LIN {X 0,Y 410.242,Z 474.921,A -85,B 0,C 180,E1 -10420.429,E2 -10420.429} C_VEL
LIN {X 0,Y 410.19,Z 477.706,A -85,B 0,C 180,E1 -10422.905,E2 -10422.905} C_VEL
LIN {X 0,Y 413.022,Z 490.224,A -85,B 0,C 180,E1 -10423.479,E2 -10423.479} C_VEL
LIN {X 0,Y 414.798,Z 499.639,A -85,B 0,C 180,E1 -10424.015,E2 -10424.015} C_VEL
LIN {X 0,Y 414.098,Z 513.044,A -85,B 0,C 180,E1 -10424.874,E2 -10424.874} C_VEL
LIN {X 0,Y 413.502,Z 524.652,A -85,B 0,C 180,E1 -10425.839,E2 -10425.839} C_VEL
LIN {X 0,Y 412.71,Z 536.519,A -85,B 0,C 180,E1 -10427.085,E2 -10427.085} C_VEL
LIN {X 0,Y 412.094,Z 545.096,A -85,B 0,C 180,E1 -10428.191,E2 -10428.191} C_VEL
LIN {X 0,Y 411.578,Z 553.045,A -85,B 0,C 180,E1 -10429.422,E2 -10429.422} C_VEL
LIN {X 0,Y 411.062,Z 560.821,A -85,B 0,C 180,E1 -10430.9,E2 -10430.9} C_VEL
LIN {X 0,Y 410.649,Z 568.02,A -85,B 0,C 180,E1 -10432.626,E2 -10432.626} C_VEL
LIN {X 0,Y 410.417,Z 572.805,A -85,B 0,C 180,E1 -10434.103,E2 -10434.103} C_VEL
LIN {X 0,Y 410.245,Z 576.463,A -85,B 0,C 180,E1 -10435.578,E2 -10435.578} C_VEL
LIN {X 0,Y 410.203,Z 579.083,A -85,B 0,C 180,E1 -10437.054,E2 -10437.054} C_VEL
LIN {X 0,Y 410.105,Z 580.298,A -85,B 0,C 180,E1 -10438.036,E2 -10438.036} C_VEL
LIN {X 0,Y 410.034,Z 581.469,A -85,B 0,C 180,E1 -10440,E2 -10440} C_VEL
LIN {X 0,Y 410.098,Z 581.463,A -85,B 0,C 180,E1 -10440.982,E2 -10440.982} C_VEL
LIN {X 0,Y 410.164,Z 581.016,A -85,B 0,C 180,E1 -10441.964,E2 -10441.964} C_VEL
LIN {X 0,Y 410.37,Z 578.907,A -85,B 0,C 180,E1 -10443.928,E2 -10443.928} C_VEL
LIN {X 0,Y 410.407,Z 576.222,A -85,B 0,C 180,E1 -10445.404,E2 -10445.404} C_VEL
LIN {X 0,Y 410.821,Z 571.701,A -85,B 0,C 180,E1 -10447.15,E2 -10447.15} C_VEL
LIN {X 0,Y 411.288,Z 565.724,A -85,B 0,C 180,E1 -10448.846,E2 -10448.846} C_VEL
LIN {X 0,Y 411.884,Z 559.118,A -85,B 0,C 180,E1 -10450.321,E2 -10450.321} C_VEL
LIN {X 0,Y 412.549,Z 550.966,A -85,B 0,C 180,E1 -10451.796,E2 -10451.796} C_VEL
LIN {X 0,Y 413.277,Z 542.616,A -85,B 0,C 180,E1 -10453.022,E2 -10453.022} C_VEL
LIN {X 0,Y 414.292,Z 531.763,A -85,B 0,C 180,E1 -10454.315,E2 -10454.315} C_VEL
LIN {X 0,Y 415.018,Z 521.116,A -85,B 0,C 180,E1 -10455.343,E2 -10455.343} C_VEL
LIN {X 0,Y 415.909,Z 508.281,A -85,B 0,C 180,E1 -10456.316,E2 -10456.316} C_VEL
LIN {X 0,Y 416.336,Z 500.964,A -85,B 0,C 180,E1 -10456.767,E2 -10456.767} C_VEL
LIN {X 0,Y 414.23,Z 492.241,A -85,B 0,C 180,E1 -10457.376,E2 -10457.376} C_VEL
LIN {X 0,Y 410.7,Z 481.456,A -85,B 0,C 180,E1 -10458.069,E2 -10458.069} C_VEL
LIN {X 0,Y 410.796,Z 479.163,A -85,B 0,C 180,E1 -10461.056,E2 -10461.056} C_VEL
LIN {X 0,Y 411.017,Z 476.941,A -85,B 0,C 180,E1 -10464.228,E2 -10464.228} C_VEL
LIN {X 0,Y 411.243,Z 474.906,A -85,B 0,C 180,E1 -10467.479,E2 -10467.479} C_VEL
LIN {X 0,Y 411.549,Z 473.168,A -85,B 0,C 180,E1 -10470.818,E2 -10470.818} C_VEL
LIN {X 0,Y 411.822,Z 472.142,A -85,B 0,C 180,E1 -10473.257,E2 -10473.257} C_VEL
LIN {X 0,Y 412.004,Z 471.503,A -85,B 0,C 180,E1 -10475.449,E2 -10475.449} C_VEL
LIN {X 0,Y 412.143,Z 471.083,A -85,B 0,C 180,E1 -10478.334,E2 -10478.334} C_VEL
LIN {X 0,Y 412.263,Z 471.372,A -85,B 0,C 180,E1 -10481.671,E2 -10481.671} C_VEL
LIN {X 0,Y 412.44,Z 472.28,A -85,B 0,C 180,E1 -10484.318,E2 -10484.318} C_VEL
LIN {X 0,Y 412.772,Z 473.906,A -85,B 0,C 180,E1 -10487.074,E2 -10487.074} C_VEL
LIN {X 0,Y 413.164,Z 476.415,A -85,B 0,C 180,E1 -10489.948,E2 -10489.948} C_VEL
LIN {X 0,Y 413.547,Z 479.076,A -85,B 0,C 180,E1 -10492.28,E2 -10492.28} C_VEL
LIN {X 0,Y 413.475,Z 482.47,A -85,B 0,C 180,E1 -10494.674,E2 -10494.674} C_VEL
LIN {X 0,Y 412.817,Z 487.359,A -85,B 0,C 180,E1 -10497.57,E2 -10497.57} C_VEL
LIN {X 0,Y 412.015,Z 493.889,A -85,B 0,C 180,E1 -10500.946,E2 -10500.946} C_VEL
LIN {X 0,Y 411.478,Z 500.74,A -85,B 0,C 180,E1 -10504.18,E2 -10504.18} C_VEL
LIN {X 0,Y 410.945,Z 509.273,A -85,B 0,C 180,E1 -10507.899,E2 -10507.899} C_VEL
LIN {X 0,Y 410.585,Z 516.838,A -85,B 0,C 180,E1 -10511.021,E2 -10511.021} C_VEL
LIN {X 0,Y 410.509,Z 518.931,A -85,B 0,C 180,E1 -10511.858,E2 -10511.858} C_VEL
LIN {X 0,Y 413.253,Z 533.559,A -85,B 0,C 180,E1 -10512.6,E2 -10512.6} C_VEL
LIN {X 0,Y 414.423,Z 546.638,A -85,B 0,C 180,E1 -10513.371,E2 -10513.371} C_VEL
LIN {X 0,Y 414.678,Z 554.233,A -85,B 0,C 180,E1 -10513.887,E2 -10513.887} C_VEL
LIN {X 0,Y 413.747,Z 566.78,A -85,B 0,C 180,E1 -10514.861,E2 -10514.861} C_VEL
LIN {X 0,Y 412.777,Z 578.942,A -85,B 0,C 180,E1 -10516.046,E2 -10516.046} C_VEL
LIN {X 0,Y 411.95,Z 588.41,A -85,B 0,C 180,E1 -10517.186,E2 -10517.186} C_VEL
LIN {X 0,Y 411.266,Z 598.435,A -85,B 0,C 180,E1 -10518.666,E2 -10518.666} C_VEL
LIN {X 0,Y 410.729,Z 606.584,A -85,B 0,C 180,E1 -10520.147,E2 -10520.147} C_VEL
LIN {X 0,Y 410.367,Z 613.151,A -85,B 0,C 180,E1 -10521.629,E2 -10521.629} C_VEL
LIN {X 0,Y 410.163,Z 618.42,A -85,B 0,C 180,E1 -10523.111,E2 -10523.111} C_VEL
LIN {X 0,Y 410.042,Z 622.525,A -85,B 0,C 180,E1 -10524.591,E2 -10524.591} C_VEL
LIN {X 0,Y 409.979,Z 625.565,A -85,B 0,C 180,E1 -10526.068,E2 -10526.068} C_VEL
LIN {X 0,Y 410.045,Z 627.027,A -85,B 0,C 180,E1 -10527.053,E2 -10527.053} C_VEL
LIN {X 0,Y 410.059,Z 628.075,A -85,B 0,C 180,E1 -10528.036,E2 -10528.036} C_VEL
LIN {X 0,Y 410.026,Z 628.699,A -85,B 0,C 180,E1 -10529.018,E2 -10529.018} C_VEL
LIN {X 0,Y 410.047,Z 628.867,A -85,B 0,C 180,E1 -10530,E2 -10530} C_VEL
LIN {X 0,Y 410.037,Z 628.623,A -85,B 0,C 180,E1 -10530.982,E2 -10530.982} C_VEL
LIN {X 0,Y 410.058,Z 627.976,A -85,B 0,C 180,E1 -10531.964,E2 -10531.964} C_VEL
LIN {X 0,Y 410.07,Z 626.896,A -85,B 0,C 180,E1 -10532.947,E2 -10532.947} C_VEL
LIN {X 0,Y 409.976,Z 625.339,A -85,B 0,C 180,E1 -10533.932,E2 -10533.932} C_VEL
LIN {X 0,Y 410.079,Z 622.192,A -85,B 0,C 180,E1 -10535.409,E2 -10535.409} C_VEL
LIN {X 0,Y 410.163,Z 617.933,A -85,B 0,C 180,E1 -10536.889,E2 -10536.889} C_VEL
LIN {X 0,Y 410.402,Z 611.438,A -85,B 0,C 180,E1 -10538.618,E2 -10538.618} C_VEL
LIN {X 0,Y 410.759,Z 604.31,A -85,B 0,C 180,E1 -10540.1,E2 -10540.1} C_VEL
LIN {X 0,Y 411.341,Z 595.431,A -85,B 0,C 180,E1 -10541.581,E2 -10541.581} C_VEL
LIN {X 0,Y 411.912,Z 586.362,A -85,B 0,C 180,E1 -10542.815,E2 -10542.815} C_VEL
LIN {X 0,Y 412.686,Z 575.411,A -85,B 0,C 180,E1 -10544.019,E2 -10544.019} C_VEL
LIN {X 0,Y 413.372,Z 563.98,A -85,B 0,C 180,E1 -10545.027,E2 -10545.027} C_VEL
LIN {X 0,Y 414.125,Z 551.921,A -85,B 0,C 180,E1 -10545.861,E2 -10545.861} C_VEL
LIN {X 0,Y 412.917,Z 539.848,A -85,B 0,C 180,E1 -10546.548,E2 -10546.548} C_VEL
LIN {X 0,Y 410.997,Z 525.799,A -85,B 0,C 180,E1 -10547.153,E2 -10547.153} C_VEL
LIN {X 0,Y 410.521,Z 522.375,A -85,B 0,C 180,E1 -10547.266,E2 -10547.266} C_VEL
LIN {X 0,Y 410.805,Z 514.358,A -85,B 0,C 180,E1 -10550.531,E2 -10550.531} C_VEL
LIN {X 0,Y 411.209,Z 506.721,A -85,B 0,C 180,E1 -10553.681,E2 -10553.681} C_VEL
LIN {X 0,Y 411.736,Z 499.086,A -85,B 0,C 180,E1 -10556.893,E2 -10556.893} C_VEL
LIN {X 0,Y 412.268,Z 491.444,A -85,B 0,C 180,E1 -10560.191,E2 -10560.191} C_VEL
LIN {X 0,Y 412.923,Z 483.99,A -85,B 0,C 180,E1 -10563.489,E2 -10563.489} C_VEL
LIN {X 0,Y 413.34,Z 478.666,A -85,B 0,C 180,E1 -10565.916,E2 -10565.916} C_VEL
LIN {X 0,Y 412.708,Z 473.491,A -85,B 0,C 180,E1 -10568.433,E2 -10568.433} C_VEL
LIN {X 0,Y 411.547,Z 466.979,A -85,B 0,C 180,E1 -10571.759,E2 -10571.759} C_VEL
LIN {X 0,Y 411.244,Z 465.261,A -85,B 0,C 180,E1 -10572.705,E2 -10572.705} C_VEL
LIN {X 0,Y 411.237,Z 465.262,A -85,B 0,C 180,E1 -10575.871,E2 -10575.871} C_VEL
LIN {X 0,Y 411.206,Z 465.265,A -85,B 0,C 180,E1 -10578.765,E2 -10578.765} C_VEL
LIN {X 0,Y 411.194,Z 465.264,A -85,B 0,C 180,E1 -10582.026,E2 -10582.026} C_VEL
LIN {X 0,Y 411.207,Z 465.262,A -85,B 0,C 180,E1 -10585.667,E2 -10585.667} C_VEL
LIN {X 0,Y 411.191,Z 465.265,A -85,B 0,C 180,E1 -10589.152,E2 -10589.152} C_VEL
LIN {X 0,Y 411.26,Z 465.258,A -85,B 0,C 180,E1 -10592.522,E2 -10592.522} C_VEL
LIN {X 0,Y 411.228,Z 465.258,A -85,B 0,C 180,E1 -10595.785,E2 -10595.785} C_VEL
LIN {X 0,Y 411.198,Z 465.266,A -85,B 0,C 180,E1 -10598.966,E2 -10598.966} C_VEL
LIN {X 0,Y 411.255,Z 465.257,A -85,B 0,C 180,E1 -10602.085,E2 -10602.085} C_VEL
LIN {X 0,Y 411.262,Z 465.257,A -85,B 0,C 180,E1 -10605.148,E2 -10605.148} C_VEL
LIN {X 0,Y 411.286,Z 465.254,A -85,B 0,C 180,E1 -10608.167,E2 -10608.167} C_VEL
LIN {X 0,Y 411.484,Z 465.23,A -85,B 0,C 180,E1 -10612.147,E2 -10612.147} C_VEL
LIN {X 0,Y 411.477,Z 465.231,A -85,B 0,C 180,E1 -10614.118,E2 -10614.118} C_VEL
LIN {X 0,Y 411.513,Z 465.225,A -85,B 0,C 180,E1 -10618.043,E2 -10618.043} C_VEL
LIN {X 0,Y 411.645,Z 465.21,A -85,B 0,C 180,E1 -10620,E2 -10620} C_VEL
LIN {X 0,Y 411.467,Z 465.231,A -85,B 0,C 180,E1 -10622.937,E2 -10622.937} C_VEL
LIN {X 0,Y 411.463,Z 465.232,A -85,B 0,C 180,E1 -10626.867,E2 -10626.867} C_VEL
LIN {X 0,Y 411.296,Z 465.252,A -85,B 0,C 180,E1 -10629.839,E2 -10629.839} C_VEL
LIN {X 0,Y 411.308,Z 465.25,A -85,B 0,C 180,E1 -10633.104,E2 -10633.104} C_VEL
LIN {X 0,Y 411.265,Z 465.257,A -85,B 0,C 180,E1 -10636.869,E2 -10636.869} C_VEL
LIN {X 0,Y 411.233,Z 465.261,A -85,B 0,C 180,E1 -10639.987,E2 -10639.987} C_VEL
LIN {X 0,Y 411.206,Z 465.263,A -85,B 0,C 180,E1 -10643.148,E2 -10643.148} C_VEL
LIN {X 0,Y 411.24,Z 465.262,A -85,B 0,C 180,E1 -10646.381,E2 -10646.381} C_VEL
LIN {X 0,Y 411.203,Z 465.264,A -85,B 0,C 180,E1 -10649.713,E2 -10649.713} C_VEL
LIN {X 0,Y 411.209,Z 465.26,A -85,B 0,C 180,E1 -10653.156,E2 -10653.156} C_VEL
LIN {X 0,Y 411.198,Z 465.266,A -85,B 0,C 180,E1 -10656.553,E2 -10656.553} C_VEL
LIN {X 0,Y 411.214,Z 465.262,A -85,B 0,C 180,E1 -10659.728,E2 -10659.728} C_VEL
LIN {X 0,Y 411.181,Z 465.266,A -85,B 0,C 180,E1 -10663.133,E2 -10663.133} C_VEL
LIN {X 0,Y 411.173,Z 465.268,A -85,B 0,C 180,E1 -10665.881,E2 -10665.881} C_VEL
LIN {X 0,Y 411.167,Z 465.268,A -85,B 0,C 180,E1 -10668.772,E2 -10668.772} C_VEL
LIN {X 0,Y 411.204,Z 465.265,A -85,B 0,C 180,E1 -10672.027,E2 -10672.027} C_VEL
LIN {X 0,Y 411.21,Z 465.262,A -85,B 0,C 180,E1 -10675.667,E2 -10675.667} C_VEL
LIN {X 0,Y 411.193,Z 465.264,A -85,B 0,C 180,E1 -10679.153,E2 -10679.153} C_VEL
LIN {X 0,Y 411.262,Z 465.256,A -85,B 0,C 180,E1 -10682.523,E2 -10682.523} C_VEL
LIN {X 0,Y 411.231,Z 465.262,A -85,B 0,C 180,E1 -10685.785,E2 -10685.785} C_VEL
LIN {X 0,Y 411.201,Z 465.262,A -85,B 0,C 180,E1 -10688.966,E2 -10688.966} C_VEL
LIN {X 0,Y 411.255,Z 465.259,A -85,B 0,C 180,E1 -10692.085,E2 -10692.085} C_VEL
LIN {X 0,Y 411.264,Z 465.255,A -85,B 0,C 180,E1 -10695.148,E2 -10695.148} C_VEL
LIN {X 0,Y 411.288,Z 465.255,A -85,B 0,C 180,E1 -10698.167,E2 -10698.167} C_VEL
LIN {X 0,Y 411.356,Z 465.244,A -85,B 0,C 180,E1 -10701.155,E2 -10701.155} C_VEL
LIN {X 0,Y 411.463,Z 465.234,A -85,B 0,C 180,E1 -10704.118,E2 -10704.118} C_VEL
LIN {X 0,Y 411.517,Z 465.226,A -85,B 0,C 180,E1 -10708.043,E2 -10708.043} C_VEL
LIN {X 0,Y 411.645,Z 465.211,A -85,B 0,C 180,E1 -10710,E2 -10710} C_VEL
LIN {X 0,Y 411.462,Z 465.23,A -85,B 0,C 180,E1 -10712.937,E2 -10712.937} C_VEL
LIN {X 0,Y 411.476,Z 465.231,A -85,B 0,C 180,E1 -10715.882,E2 -10715.882} C_VEL
LIN {X 0,Y 411.356,Z 465.243,A -85,B 0,C 180,E1 -10718.845,E2 -10718.845} C_VEL
LIN {X 0,Y 411.289,Z 465.254,A -85,B 0,C 180,E1 -10721.833,E2 -10721.833} C_VEL
LIN {X 0,Y 411.265,Z 465.254,A -85,B 0,C 180,E1 -10724.853,E2 -10724.853} C_VEL
LIN {X 0,Y 411.244,Z 465.257,A -85,B 0,C 180,E1 -10727.586,E2 -10727.586} C_VEL
LIN {X 0,Y 410.584,Z 465.343,A -85,B 0,C 180,E1 -10728.404,E2 -10728.404} C_VEL
LIN {X 0,Y 407.696,Z 465.704,A -85,B 0,C 180,E1 -10729.732,E2 -10729.732} C_VEL
LIN {X 0,Y 405.253,Z 466.005,A -85,B 0,C 180,E1 -10730.805,E2 -10730.805} C_VEL
LIN {X 0,Y 404.217,Z 466.135,A -85,B 0,C 180,E1 -10731.635,E2 -10731.635} C_VEL
LIN {X 0,Y 404.141,Z 466.14,A -85,B 0,C 180,E1 -10731.916,E2 -10731.916} C_VEL
LIN {X 0,Y 404.22,Z 466.134,A -85,B 0,C 180,E1 -10735.297,E2 -10735.297} C_VEL
LIN {X 0,Y 404.2,Z 466.139,A -85,B 0,C 180,E1 -10738,E2 -10738} C_VEL
LIN {X 0,Y 404.144,Z 466.145,A -85,B 0,C 180,E1 -10741.558,E2 -10741.558} C_VEL
LIN {X 0,Y 404.189,Z 466.137,A -85,B 0,C 180,E1 -10745.016,E2 -10745.016} C_VEL
LIN {X 0,Y 404.162,Z 466.139,A -85,B 0,C 180,E1 -10748.756,E2 -10748.756} C_VEL
LIN {X 0,Y 404.127,Z 466.146,A -85,B 0,C 180,E1 -10751.6,E2 -10751.6} C_VEL
LIN {X 0,Y 404.149,Z 466.14,A -85,B 0,C 180,E1 -10754.522,E2 -10754.522} C_VEL
LIN {X 0,Y 404.14,Z 466.145,A -85,B 0,C 180,E1 -10757.296,E2 -10757.296} C_VEL
LIN {X 0,Y 404.172,Z 466.142,A -85,B 0,C 180,E1 -10759.955,E2 -10759.955} C_VEL
LIN {X 0,Y 404.123,Z 466.145,A -85,B 0,C 180,E1 -10763.128,E2 -10763.128} C_VEL
LIN {X 0,Y 404.049,Z 466.154,A -85,B 0,C 180,E1 -10764.97,E2 -10764.97} C_VEL
LIN {X 0,Y 403.66,Z 466.204,A -85,B 0,C 180,E1 -10768.554,E2 -10768.554} C_VEL
LIN {X 0,Y 403.415,Z 466.238,A -85,B 0,C 180,E1 -10770.804,E2 -10770.804} C_VEL
LIN {X 0,Y 403.339,Z 468.056,A -85,B 0,C 180,E1 -10773.061,E2 -10773.061} C_VEL
LIN {X 0,Y 403.256,Z 470.252,A -85,B 0,C 180,E1 -10775.274,E2 -10775.274} C_VEL
LIN {X 0,Y 403.144,Z 473.565,A -85,B 0,C 180,E1 -10778.525,E2 -10778.525} C_VEL
LIN {X 0,Y 403.155,Z 475.779,A -85,B 0,C 180,E1 -10780.657,E2 -10780.657} C_VEL
LIN {X 0,Y 403.121,Z 477.917,A -85,B 0,C 180,E1 -10782.662,E2 -10782.662} C_VEL
LIN {X 0,Y 405.962,Z 490.643,A -85,B 0,C 180,E1 -10783.25,E2 -10783.25} C_VEL
LIN {X 0,Y 407.853,Z 500.898,A -85,B 0,C 180,E1 -10783.849,E2 -10783.849} C_VEL
LIN {X 0,Y 407.106,Z 514.287,A -85,B 0,C 180,E1 -10784.736,E2 -10784.736} C_VEL
LIN {X 0,Y 406.536,Z 525.173,A -85,B 0,C 180,E1 -10785.67,E2 -10785.67} C_VEL
LIN {X 0,Y 405.767,Z 536.345,A -85,B 0,C 180,E1 -10786.86,E2 -10786.86} C_VEL
LIN {X 0,Y 405.017,Z 546.743,A -85,B 0,C 180,E1 -10788.235,E2 -10788.235} C_VEL
LIN {X 0,Y 404.399,Z 555.835,A -85,B 0,C 180,E1 -10789.739,E2 -10789.739} C_VEL
LIN {X 0,Y 403.892,Z 563.194,A -85,B 0,C 180,E1 -10791.242,E2 -10791.242} C_VEL
LIN {X 0,Y 403.607,Z 568.167,A -85,B 0,C 180,E1 -10792.496,E2 -10792.496} C_VEL
LIN {X 0,Y 403.36,Z 573.012,A -85,B 0,C 180,E1 -10793.999,E2 -10793.999} C_VEL
LIN {X 0,Y 403.16,Z 576.726,A -85,B 0,C 180,E1 -10795.501,E2 -10795.501} C_VEL
LIN {X 0,Y 403.139,Z 579.398,A -85,B 0,C 180,E1 -10797.002,E2 -10797.002} C_VEL
LIN {X 0,Y 403.035,Z 580.663,A -85,B 0,C 180,E1 -10798.001,E2 -10798.001} C_VEL
LIN {X 0,Y 402.953,Z 581.89,A -85,B 0,C 180,E1 -10800,E2 -10800} C_VEL
LIN {X 0,Y 403.018,Z 581.912,A -85,B 0,C 180,E1 -10800.999,E2 -10800.999} C_VEL
LIN {X 0,Y 403.09,Z 581.508,A -85,B 0,C 180,E1 -10801.998,E2 -10801.998} C_VEL
LIN {X 0,Y 403.324,Z 579.443,A -85,B 0,C 180,E1 -10803.997,E2 -10803.997} C_VEL
LIN {X 0,Y 403.354,Z 576.8,A -85,B 0,C 180,E1 -10805.499,E2 -10805.499} C_VEL
LIN {X 0,Y 403.803,Z 572.489,A -85,B 0,C 180,E1 -10807.224,E2 -10807.224} C_VEL
LIN {X 0,Y 404.308,Z 566.458,A -85,B 0,C 180,E1 -10809,E2 -10809} C_VEL
LIN {X 0,Y 404.95,Z 559.945,A -85,B 0,C 180,E1 -10810.5,E2 -10810.5} C_VEL
LIN {X 0,Y 405.661,Z 551.887,A -85,B 0,C 180,E1 -10811.999,E2 -10811.999} C_VEL
LIN {X 0,Y 406.444,Z 543.623,A -85,B 0,C 180,E1 -10813.245,E2 -10813.245} C_VEL
LIN {X 0,Y 407.529,Z 532.805,A -85,B 0,C 180,E1 -10814.569,E2 -10814.569} C_VEL
LIN {X 0,Y 408.309,Z 522.565,A -85,B 0,C 180,E1 -10815.601,E2 -10815.601} C_VEL
LIN {X 0,Y 409.249,Z 510.108,A -85,B 0,C 180,E1 -10816.589,E2 -10816.589} C_VEL
LIN {X 0,Y 409.745,Z 502.76,A -85,B 0,C 180,E1 -10817.067,E2 -10817.067} C_VEL
LIN {X 0,Y 407.618,Z 493.899,A -85,B 0,C 180,E1 -10817.71,E2 -10817.71} C_VEL
LIN {X 0,Y 403.693,Z 482.076,A -85,B 0,C 180,E1 -10818.525,E2 -10818.525} C_VEL
LIN {X 0,Y 403.788,Z 479.932,A -85,B 0,C 180,E1 -10821.439,E2 -10821.439} C_VEL
LIN {X 0,Y 404.029,Z 477.77,A -85,B 0,C 180,E1 -10824.675,E2 -10824.675} C_VEL
LIN {X 0,Y 404.279,Z 475.811,A -85,B 0,C 180,E1 -10827.993,E2 -10827.993} C_VEL
LIN {X 0,Y 404.629,Z 474.173,A -85,B 0,C 180,E1 -10831.404,E2 -10831.404} C_VEL
LIN {X 0,Y 404.873,Z 473.332,A -85,B 0,C 180,E1 -10833.743,E2 -10833.743} C_VEL
LIN {X 0,Y 405.08,Z 472.757,A -85,B 0,C 180,E1 -10836.149,E2 -10836.149} C_VEL
LIN {X 0,Y 405.203,Z 472.55,A -85,B 0,C 180,E1 -10838.693,E2 -10838.693} C_VEL
LIN {X 0,Y 405.355,Z 472.927,A -85,B 0,C 180,E1 -10841.795,E2 -10841.795} C_VEL
LIN {X 0,Y 405.62,Z 474.313,A -85,B 0,C 180,E1 -10845.267,E2 -10845.267} C_VEL
LIN {X 0,Y 405.964,Z 476.262,A -85,B 0,C 180,E1 -10848.109,E2 -10848.109} C_VEL
LIN {X 0,Y 406.502,Z 479.632,A -85,B 0,C 180,E1 -10851.508,E2 -10851.508} C_VEL
LIN {X 0,Y 406.623,Z 481.2,A -85,B 0,C 180,E1 -10852.776,E2 -10852.776} C_VEL
LIN {X 0,Y 406.398,Z 484.692,A -85,B 0,C 180,E1 -10855.202,E2 -10855.202} C_VEL
LIN {X 0,Y 405.716,Z 489.579,A -85,B 0,C 180,E1 -10858.082,E2 -10858.082} C_VEL
LIN {X 0,Y 404.887,Z 496.099,A -85,B 0,C 180,E1 -10861.488,E2 -10861.488} C_VEL
LIN {X 0,Y 404.352,Z 502.758,A -85,B 0,C 180,E1 -10864.663,E2 -10864.663} C_VEL
LIN {X 0,Y 403.814,Z 511.578,A -85,B 0,C 180,E1 -10868.562,E2 -10868.562} C_VEL
LIN {X 0,Y 403.482,Z 518.346,A -85,B 0,C 180,E1 -10871.399,E2 -10871.399} C_VEL
LIN {X 0,Y 406.164,Z 531.761,A -85,B 0,C 180,E1 -10872.117,E2 -10872.117} C_VEL
LIN {X 0,Y 407.317,Z 542.322,A -85,B 0,C 180,E1 -10872.744,E2 -10872.744} C_VEL
LIN {X 0,Y 407.9,Z 554.877,A -85,B 0,C 180,E1 -10873.612,E2 -10873.612} C_VEL
LIN {X 0,Y 406.906,Z 567.099,A -85,B 0,C 180,E1 -10874.6,E2 -10874.6} C_VEL
LIN {X 0,Y 405.935,Z 578.273,A -85,B 0,C 180,E1 -10875.717,E2 -10875.717} C_VEL
LIN {X 0,Y 405.004,Z 588.378,A -85,B 0,C 180,E1 -10876.962,E2 -10876.962} C_VEL
LIN {X 0,Y 404.293,Z 598.314,A -85,B 0,C 180,E1 -10878.468,E2 -10878.468} C_VEL
LIN {X 0,Y 403.689,Z 606.372,A -85,B 0,C 180,E1 -10879.974,E2 -10879.974} C_VEL
LIN {X 0,Y 403.324,Z 612.89,A -85,B 0,C 180,E1 -10881.482,E2 -10881.482} C_VEL
LIN {X 0,Y 403.075,Z 618.117,A -85,B 0,C 180,E1 -10882.989,E2 -10882.989} C_VEL
LIN {X 0,Y 402.942,Z 622.187,A -85,B 0,C 180,E1 -10884.495,E2 -10884.495} C_VEL
LIN {X 0,Y 402.897,Z 625.201,A -85,B 0,C 180,E1 -10885.999,E2 -10885.999} C_VEL
LIN {X 0,Y 402.943,Z 626.649,A -85,B 0,C 180,E1 -10887.001,E2 -10887.001} C_VEL
LIN {X 0,Y 402.987,Z 627.685,A -85,B 0,C 180,E1 -10888.001,E2 -10888.001} C_VEL
LIN {X 0,Y 402.949,Z 628.281,A -85,B 0,C 180,E1 -10889.001,E2 -10889.001} C_VEL
LIN {X 0,Y 402.965,Z 628.432,A -85,B 0,C 180,E1 -10890,E2 -10890} C_VEL
LIN {X 0,Y 402.959,Z 628.174,A -85,B 0,C 180,E1 -10890.999,E2 -10890.999} C_VEL
LIN {X 0,Y 402.987,Z 627.511,A -85,B 0,C 180,E1 -10891.999,E2 -10891.999} C_VEL
LIN {X 0,Y 402.971,Z 626.39,A -85,B 0,C 180,E1 -10892.999,E2 -10892.999} C_VEL
LIN {X 0,Y 402.896,Z 624.815,A -85,B 0,C 180,E1 -10894.001,E2 -10894.001} C_VEL
LIN {X 0,Y 402.998,Z 621.622,A -85,B 0,C 180,E1 -10895.504,E2 -10895.504} C_VEL
LIN {X 0,Y 403.075,Z 617.312,A -85,B 0,C 180,E1 -10897.01,E2 -10897.01} C_VEL
LIN {X 0,Y 403.351,Z 610.761,A -85,B 0,C 180,E1 -10898.769,E2 -10898.769} C_VEL
LIN {X 0,Y 403.711,Z 603.543,A -85,B 0,C 180,E1 -10900.279,E2 -10900.279} C_VEL
LIN {X 0,Y 404.356,Z 594.597,A -85,B 0,C 180,E1 -10901.784,E2 -10901.784} C_VEL
LIN {X 0,Y 404.956,Z 585.444,A -85,B 0,C 180,E1 -10903.039,E2 -10903.039} C_VEL
LIN {X 0,Y 405.66,Z 575.352,A -85,B 0,C 180,E1 -10904.165,E2 -10904.165} C_VEL
LIN {X 0,Y 406.358,Z 564.32,A -85,B 0,C 180,E1 -10905.164,E2 -10905.164} C_VEL
LIN {X 0,Y 407.155,Z 552.212,A -85,B 0,C 180,E1 -10906.032,E2 -10906.032} C_VEL
LIN {X 0,Y 405.767,Z 538.968,A -85,B 0,C 180,E1 -10906.804,E2 -10906.804} C_VEL
LIN {X 0,Y 403.826,Z 525.012,A -85,B 0,C 180,E1 -10907.416,E2 -10907.416} C_VEL
LIN {X 0,Y 403.459,Z 522.002,A -85,B 0,C 180,E1 -10907.532,E2 -10907.532} C_VEL
LIN {X 0,Y 403.771,Z 513.899,A -85,B 0,C 180,E1 -10910.905,E2 -10910.905} C_VEL
LIN {X 0,Y 404.303,Z 505.031,A -85,B 0,C 180,E1 -10914.657,E2 -10914.657} C_VEL
LIN {X 0,Y 404.859,Z 497.426,A -85,B 0,C 180,E1 -10917.95,E2 -10917.95} C_VEL
LIN {X 0,Y 405.445,Z 489.784,A -85,B 0,C 180,E1 -10921.334,E2 -10921.334} C_VEL
LIN {X 0,Y 406.072,Z 483.349,A -85,B 0,C 180,E1 -10924.259,E2 -10924.259} C_VEL
LIN {X 0,Y 406.317,Z 479.589,A -85,B 0,C 180,E1 -10926.022,E2 -10926.022} C_VEL
LIN {X 0,Y 405.651,Z 474.386,A -85,B 0,C 180,E1 -10928.587,E2 -10928.587} C_VEL
LIN {X 0,Y 404.616,Z 468.458,A -85,B 0,C 180,E1 -10931.678,E2 -10931.678} C_VEL
LIN {X 0,Y 404.168,Z 466.142,A -85,B 0,C 180,E1 -10933.005,E2 -10933.005} C_VEL
LIN {X 0,Y 404.21,Z 466.137,A -85,B 0,C 180,E1 -10935.935,E2 -10935.935} C_VEL
LIN {X 0,Y 404.161,Z 466.142,A -85,B 0,C 180,E1 -10938.64,E2 -10938.64} C_VEL
LIN {X 0,Y 404.153,Z 466.14,A -85,B 0,C 180,E1 -10941.493,E2 -10941.493} C_VEL
LIN {X 0,Y 404.186,Z 466.14,A -85,B 0,C 180,E1 -10944.984,E2 -10944.984} C_VEL
LIN {X 0,Y 404.143,Z 466.146,A -85,B 0,C 180,E1 -10948.554,E2 -10948.554} C_VEL
LIN {X 0,Y 404.197,Z 466.136,A -85,B 0,C 180,E1 -10952,E2 -10952} C_VEL
LIN {X 0,Y 404.178,Z 466.137,A -85,B 0,C 180,E1 -10955.334,E2 -10955.334} C_VEL
LIN {X 0,Y 404.14,Z 466.145,A -85,B 0,C 180,E1 -10958.581,E2 -10958.581} C_VEL
LIN {X 0,Y 404.212,Z 466.133,A -85,B 0,C 180,E1 -10961.762,E2 -10961.762} C_VEL
LIN {X 0,Y 404.208,Z 466.136,A -85,B 0,C 180,E1 -10964.882,E2 -10964.882} C_VEL
LIN {X 0,Y 404.258,Z 466.129,A -85,B 0,C 180,E1 -10967.959,E2 -10967.959} C_VEL
LIN {X 0,Y 404.435,Z 466.108,A -85,B 0,C 180,E1 -10972.1,E2 -10972.1} C_VEL
LIN {X 0,Y 404.426,Z 466.109,A -85,B 0,C 180,E1 -10974.015,E2 -10974.015} C_VEL
LIN {X 0,Y 404.482,Z 466.1,A -85,B 0,C 180,E1 -10978.009,E2 -10978.009} C_VEL
LIN {X 0,Y 404.614,Z 466.085,A -85,B 0,C 180,E1 -10980,E2 -10980} C_VEL
LIN {X 0,Y 404.424,Z 466.108,A -85,B 0,C 180,E1 -10982.989,E2 -10982.989} C_VEL
LIN {X 0,Y 404.414,Z 466.11,A -85,B 0,C 180,E1 -10986.987,E2 -10986.987} C_VEL
LIN {X 0,Y 404.261,Z 466.129,A -85,B 0,C 180,E1 -10990.012,E2 -10990.012} C_VEL
LIN {X 0,Y 404.268,Z 466.126,A -85,B 0,C 180,E1 -10993.212,E2 -10993.212} C_VEL
LIN {X 0,Y 404.218,Z 466.133,A -85,B 0,C 180,E1 -10997.007,E2 -10997.007} C_VEL
LIN {X 0,Y 404.166,Z 466.143,A -85,B 0,C 180,E1 -11000.352,E2 -11000.352} C_VEL
LIN {X 0,Y 404.172,Z 466.139,A -85,B 0,C 180,E1 -11003.575,E2 -11003.575} C_VEL
LIN {X 0,Y 404.186,Z 466.137,A -85,B 0,C 180,E1 -11005.767,E2 -11005.767} C_VEL
LIN {X 0,Y 404.198,Z 466.138,A -85,B 0,C 180,E1 -11008,E2 -11008} C_VEL
LIN {X 0,Y 404.142,Z 466.142,A -85,B 0,C 180,E1 -11011.558,E2 -11011.558} C_VEL
LIN {X 0,Y 404.188,Z 466.137,A -85,B 0,C 180,E1 -11015.016,E2 -11015.016} C_VEL
LIN {X 0,Y 404.157,Z 466.142,A -85,B 0,C 180,E1 -11018.757,E2 -11018.757} C_VEL
LIN {X 0,Y 404.127,Z 466.144,A -85,B 0,C 180,E1 -11021.6,E2 -11021.6} C_VEL
LIN {X 0,Y 404.152,Z 466.144,A -85,B 0,C 180,E1 -11024.523,E2 -11024.523} C_VEL
LIN {X 0,Y 404.141,Z 466.141,A -85,B 0,C 180,E1 -11027.296,E2 -11027.296} C_VEL
LIN {X 0,Y 404.172,Z 466.142,A -85,B 0,C 180,E1 -11029.956,E2 -11029.956} C_VEL
LIN {X 0,Y 404.143,Z 466.142,A -85,B 0,C 180,E1 -11033.125,E2 -11033.125} C_VEL
LIN {X 0,Y 404.148,Z 466.145,A -85,B 0,C 180,E1 -11036.188,E2 -11036.188} C_VEL
LIN {X 0,Y 404.149,Z 466.143,A -85,B 0,C 180,E1 -11039.715,E2 -11039.715} C_VEL
LIN {X 0,Y 404.199,Z 466.134,A -85,B 0,C 180,E1 -11043.123,E2 -11043.123} C_VEL
LIN {X 0,Y 404.181,Z 466.138,A -85,B 0,C 180,E1 -11045.335,E2 -11045.335} C_VEL
LIN {X 0,Y 404.143,Z 466.143,A -85,B 0,C 180,E1 -11048.581,E2 -11048.581} C_VEL
LIN {X 0,Y 404.213,Z 466.136,A -85,B 0,C 180,E1 -11051.762,E2 -11051.762} C_VEL
LIN {X 0,Y 404.211,Z 466.133,A -85,B 0,C 180,E1 -11054.882,E2 -11054.882} C_VEL
LIN {X 0,Y 404.261,Z 466.132,A -85,B 0,C 180,E1 -11057.959,E2 -11057.959} C_VEL
LIN {X 0,Y 404.293,Z 466.123,A -85,B 0,C 180,E1 -11060.999,E2 -11060.999} C_VEL
LIN {X 0,Y 404.41,Z 466.113,A -85,B 0,C 180,E1 -11064.015,E2 -11064.015} C_VEL
LIN {X 0,Y 404.485,Z 466.102,A -85,B 0,C 180,E1 -11068.009,E2 -11068.009} C_VEL
LIN {X 0,Y 404.614,Z 466.087,A -85,B 0,C 180,E1 -11070,E2 -11070} C_VEL
LIN {X 0,Y 404.42,Z 466.107,A -85,B 0,C 180,E1 -11072.989,E2 -11072.989} C_VEL
LIN {X 0,Y 404.423,Z 466.11,A -85,B 0,C 180,E1 -11075.985,E2 -11075.985} C_VEL
LIN {X 0,Y 404.293,Z 466.122,A -85,B 0,C 180,E1 -11079.001,E2 -11079.001} C_VEL
LIN {X 0,Y 404.261,Z 466.13,A -85,B 0,C 180,E1 -11082.041,E2 -11082.041} C_VEL
LIN {X 0,Y 404.211,Z 466.133,A -85,B 0,C 180,E1 -11085.118,E2 -11085.118} C_VEL
LIN {X 0,Y 404.215,Z 466.135,A -85,B 0,C 180,E1 -11088.238,E2 -11088.238} C_VEL
LIN {X 0,Y 404.143,Z 466.143,A -85,B 0,C 180,E1 -11091.419,E2 -11091.419} C_VEL
LIN {X 0,Y 404.141,Z 466.14,A -85,B 0,C 180,E1 -11091.916,E2 -11091.916} C_VEL
LIN {X 0,Y 403.498,Z 466.222,A -85,B 0,C 180,E1 -11092.748,E2 -11092.748} C_VEL
LIN {X 0,Y 400.666,Z 466.579,A -85,B 0,C 180,E1 -11094.099,E2 -11094.099} C_VEL
LIN {X 0,Y 398.257,Z 466.882,A -85,B 0,C 180,E1 -11095.192,E2 -11095.192} C_VEL
LIN {X 0,Y 397.222,Z 467.008,A -85,B 0,C 180,E1 -11096.036,E2 -11096.036} C_VEL
LIN {X 0,Y 397.139,Z 467.017,A -85,B 0,C 180,E1 -11096.322,E2 -11096.322} C_VEL
LIN {X 0,Y 397.126,Z 467.016,A -85,B 0,C 180,E1 -11098.544,E2 -11098.544} C_VEL
LIN {X 0,Y 397.083,Z 467.024,A -85,B 0,C 180,E1 -11102.071,E2 -11102.071} C_VEL
LIN {X 0,Y 397.123,Z 467.018,A -85,B 0,C 180,E1 -11105.503,E2 -11105.503} C_VEL
LIN {X 0,Y 397.136,Z 467.014,A -85,B 0,C 180,E1 -11108.862,E2 -11108.862} C_VEL
LIN {X 0,Y 397.073,Z 467.024,A -85,B 0,C 180,E1 -11112.267,E2 -11112.267} C_VEL
LIN {X 0,Y 397.09,Z 467.02,A -85,B 0,C 180,E1 -11115.069,E2 -11115.069} C_VEL
LIN {X 0,Y 397.07,Z 467.026,A -85,B 0,C 180,E1 -11118.021,E2 -11118.021} C_VEL
LIN {X 0,Y 397.132,Z 467.016,A -85,B 0,C 180,E1 -11121.139,E2 -11121.139} C_VEL
LIN {X 0,Y 397.009,Z 467.031,A -85,B 0,C 180,E1 -11124.519,E2 -11124.519} C_VEL
LIN {X 0,Y 396.655,Z 467.079,A -85,B 0,C 180,E1 -11127.89,E2 -11127.89} C_VEL
LIN {X 0,Y 396.301,Z 467.127,A -85,B 0,C 180,E1 -11131.391,E2 -11131.391} C_VEL
LIN {X 0,Y 396.215,Z 470.434,A -85,B 0,C 180,E1 -11134.804,E2 -11134.804} C_VEL
LIN {X 0,Y 396.097,Z 473.785,A -85,B 0,C 180,E1 -11138.123,E2 -11138.123} C_VEL
LIN {X 0,Y 396.112,Z 476.028,A -85,B 0,C 180,E1 -11140.299,E2 -11140.299} C_VEL
LIN {X 0,Y 396.049,Z 478.389,A -85,B 0,C 180,E1 -11142.425,E2 -11142.425} C_VEL
LIN {X 0,Y 399.01,Z 491.767,A -85,B 0,C 180,E1 -11143.066,E2 -11143.066} C_VEL
LIN {X 0,Y 400.914,Z 501.376,A -85,B 0,C 180,E1 -11143.649,E2 -11143.649} C_VEL
LIN {X 0,Y 400.207,Z 513.572,A -85,B 0,C 180,E1 -11144.466,E2 -11144.466} C_VEL
LIN {X 0,Y 399.539,Z 525.667,A -85,B 0,C 180,E1 -11145.511,E2 -11145.511} C_VEL
LIN {X 0,Y 398.743,Z 537.091,A -85,B 0,C 180,E1 -11146.754,E2 -11146.754} C_VEL
LIN {X 0,Y 398.036,Z 546.584,A -85,B 0,C 180,E1 -11148.026,E2 -11148.026} C_VEL
LIN {X 0,Y 397.399,Z 555.777,A -85,B 0,C 180,E1 -11149.556,E2 -11149.556} C_VEL
LIN {X 0,Y 396.874,Z 563.226,A -85,B 0,C 180,E1 -11151.086,E2 -11151.086} C_VEL
LIN {X 0,Y 396.545,Z 568.276,A -85,B 0,C 180,E1 -11152.361,E2 -11152.361} C_VEL
LIN {X 0,Y 396.304,Z 573.194,A -85,B 0,C 180,E1 -11153.892,E2 -11153.892} C_VEL
LIN {X 0,Y 396.081,Z 576.976,A -85,B 0,C 180,E1 -11155.42,E2 -11155.42} C_VEL
LIN {X 0,Y 396.076,Z 579.709,A -85,B 0,C 180,E1 -11156.948,E2 -11156.948} C_VEL
LIN {X 0,Y 395.967,Z 581.018,A -85,B 0,C 180,E1 -11157.966,E2 -11157.966} C_VEL
LIN {X 0,Y 395.89,Z 581.867,A -85,B 0,C 180,E1 -11158.983,E2 -11158.983} C_VEL
LIN {X 0,Y 395.94,Z 582.36,A -85,B 0,C 180,E1 -11161.017,E2 -11161.017} C_VEL
LIN {X 0,Y 396.018,Z 581.999,A -85,B 0,C 180,E1 -11162.034,E2 -11162.034} C_VEL
LIN {X 0,Y 396.278,Z 579.992,A -85,B 0,C 180,E1 -11164.068,E2 -11164.068} C_VEL
LIN {X 0,Y 396.308,Z 577.416,A -85,B 0,C 180,E1 -11165.597,E2 -11165.597} C_VEL
LIN {X 0,Y 396.777,Z 573.346,A -85,B 0,C 180,E1 -11167.289,E2 -11167.289} C_VEL
LIN {X 0,Y 397.166,Z 569.069,A -85,B 0,C 180,E1 -11168.651,E2 -11168.651} C_VEL
LIN {X 0,Y 397.82,Z 563.088,A -85,B 0,C 180,E1 -11170.175,E2 -11170.175} C_VEL
LIN {X 0,Y 398.502,Z 555.662,A -85,B 0,C 180,E1 -11171.701,E2 -11171.701} C_VEL
LIN {X 0,Y 399.32,Z 546.472,A -85,B 0,C 180,E1 -11173.226,E2 -11173.226} C_VEL
LIN {X 0,Y 400.472,Z 537.193,A -85,B 0,C 180,E1 -11174.462,E2 -11174.462} C_VEL
LIN {X 0,Y 401.384,Z 526.537,A -85,B 0,C 180,E1 -11175.63,E2 -11175.63} C_VEL
LIN {X 0,Y 402.343,Z 515.244,A -85,B 0,C 180,E1 -11176.621,E2 -11176.621} C_VEL
LIN {X 0,Y 403.1,Z 504.828,A -85,B 0,C 180,E1 -11177.357,E2 -11177.357} C_VEL
LIN {X 0,Y 402.161,Z 499.439,A -85,B 0,C 180,E1 -11177.771,E2 -11177.771} C_VEL
LIN {X 0,Y 398.394,Z 487.612,A -85,B 0,C 180,E1 -11178.67,E2 -11178.67} C_VEL
LIN {X 0,Y 396.691,Z 482.723,A -85,B 0,C 180,E1 -11179.032,E2 -11179.032} C_VEL
LIN {X 0,Y 396.888,Z 479.988,A -85,B 0,C 180,E1 -11182.956,E2 -11182.956} C_VEL
LIN {X 0,Y 397.123,Z 477.984,A -85,B 0,C 180,E1 -11186.259,E2 -11186.259} C_VEL
LIN {X 0,Y 397.316,Z 476.765,A -85,B 0,C 180,E1 -11188.528,E2 -11188.528} C_VEL
LIN {X 0,Y 397.726,Z 475.257,A -85,B 0,C 180,E1 -11192.013,E2 -11192.013} C_VEL
LIN {X 0,Y 397.964,Z 474.523,A -85,B 0,C 180,E1 -11194.41,E2 -11194.41} C_VEL
LIN {X 0,Y 398.2,Z 474.045,A -85,B 0,C 180,E1 -11197.418,E2 -11197.418} C_VEL
LIN {X 0,Y 398.356,Z 474.237,A -85,B 0,C 180,E1 -11200.751,E2 -11200.751} C_VEL
LIN {X 0,Y 398.536,Z 475.103,A -85,B 0,C 180,E1 -11203.696,E2 -11203.696} C_VEL
LIN {X 0,Y 398.857,Z 476.677,A -85,B 0,C 180,E1 -11206.591,E2 -11206.591} C_VEL
LIN {X 0,Y 399.214,Z 478.906,A -85,B 0,C 180,E1 -11209.355,E2 -11209.355} C_VEL
LIN {X 0,Y 399.64,Z 482.082,A -85,B 0,C 180,E1 -11212.313,E2 -11212.313} C_VEL
LIN {X 0,Y 399.542,Z 485.052,A -85,B 0,C 180,E1 -11214.516,E2 -11214.516} C_VEL
LIN {X 0,Y 398.984,Z 488.835,A -85,B 0,C 180,E1 -11216.903,E2 -11216.903} C_VEL
LIN {X 0,Y 398.238,Z 494.068,A -85,B 0,C 180,E1 -11219.853,E2 -11219.853} C_VEL
LIN {X 0,Y 397.484,Z 501.834,A -85,B 0,C 180,E1 -11223.766,E2 -11223.766} C_VEL
LIN {X 0,Y 396.842,Z 510.183,A -85,B 0,C 180,E1 -11227.619,E2 -11227.619} C_VEL
LIN {X 0,Y 396.463,Z 517.85,A -85,B 0,C 180,E1 -11230.923,E2 -11230.923} C_VEL
LIN {X 0,Y 399.354,Z 531.827,A -85,B 0,C 180,E1 -11231.705,E2 -11231.705} C_VEL
LIN {X 0,Y 400.629,Z 542.882,A -85,B 0,C 180,E1 -11232.401,E2 -11232.401} C_VEL
LIN {X 0,Y 401.123,Z 555.575,A -85,B 0,C 180,E1 -11233.327,E2 -11233.327} C_VEL
LIN {X 0,Y 400.089,Z 567.527,A -85,B 0,C 180,E1 -11234.331,E2 -11234.331} C_VEL
LIN {X 0,Y 399.068,Z 578.469,A -85,B 0,C 180,E1 -11235.466,E2 -11235.466} C_VEL
LIN {X 0,Y 398.073,Z 588.419,A -85,B 0,C 180,E1 -11236.731,E2 -11236.731} C_VEL
LIN {X 0,Y 397.326,Z 598.249,A -85,B 0,C 180,E1 -11238.263,E2 -11238.263} C_VEL
LIN {X 0,Y 396.654,Z 606.198,A -85,B 0,C 180,E1 -11239.794,E2 -11239.794} C_VEL
LIN {X 0,Y 396.283,Z 612.659,A -85,B 0,C 180,E1 -11241.33,E2 -11241.33} C_VEL
LIN {X 0,Y 396.002,Z 617.837,A -85,B 0,C 180,E1 -11242.863,E2 -11242.863} C_VEL
LIN {X 0,Y 395.849,Z 621.869,A -85,B 0,C 180,E1 -11244.396,E2 -11244.396} C_VEL
LIN {X 0,Y 395.817,Z 624.847,A -85,B 0,C 180,E1 -11245.927,E2 -11245.927} C_VEL
LIN {X 0,Y 395.843,Z 626.278,A -85,B 0,C 180,E1 -11246.947,E2 -11246.947} C_VEL
LIN {X 0,Y 395.915,Z 627.3,A -85,B 0,C 180,E1 -11247.965,E2 -11247.965} C_VEL
LIN {X 0,Y 395.874,Z 627.859,A -85,B 0,C 180,E1 -11248.983,E2 -11248.983} C_VEL
LIN {X 0,Y 395.886,Z 627.992,A -85,B 0,C 180,E1 -11250,E2 -11250} C_VEL
LIN {X 0,Y 395.883,Z 627.716,A -85,B 0,C 180,E1 -11251.017,E2 -11251.017} C_VEL
LIN {X 0,Y 395.917,Z 627.03,A -85,B 0,C 180,E1 -11252.034,E2 -11252.034} C_VEL
LIN {X 0,Y 395.875,Z 625.869,A -85,B 0,C 180,E1 -11253.053,E2 -11253.053} C_VEL
LIN {X 0,Y 395.878,Z 623.325,A -85,B 0,C 180,E1 -11254.582,E2 -11254.582} C_VEL
LIN {X 0,Y 395.914,Z 619.362,A -85,B 0,C 180,E1 -11256.24,E2 -11256.24} C_VEL
LIN {X 0,Y 396.057,Z 614.957,A -85,B 0,C 180,E1 -11257.648,E2 -11257.648} C_VEL
LIN {X 0,Y 396.412,Z 607.786,A -85,B 0,C 180,E1 -11259.439,E2 -11259.439} C_VEL
LIN {X 0,Y 396.852,Z 599.962,A -85,B 0,C 180,E1 -11260.975,E2 -11260.975} C_VEL
LIN {X 0,Y 397.471,Z 592.001,A -85,B 0,C 180,E1 -11262.25,E2 -11262.25} C_VEL
LIN {X 0,Y 398.182,Z 581.602,A -85,B 0,C 180,E1 -11263.615,E2 -11263.615} C_VEL
LIN {X 0,Y 398.999,Z 570.348,A -85,B 0,C 180,E1 -11264.797,E2 -11264.797} C_VEL
LIN {X 0,Y 399.786,Z 558.158,A -85,B 0,C 180,E1 -11265.812,E2 -11265.812} C_VEL
LIN {X 0,Y 400.109,Z 551.72,A -85,B 0,C 180,E1 -11266.257,E2 -11266.257} C_VEL
LIN {X 0,Y 398.696,Z 539.049,A -85,B 0,C 180,E1 -11267.015,E2 -11267.015} C_VEL
LIN {X 0,Y 396.868,Z 525.276,A -85,B 0,C 180,E1 -11267.637,E2 -11267.637} C_VEL
LIN {X 0,Y 396.375,Z 521.702,A -85,B 0,C 180,E1 -11267.776,E2 -11267.776} C_VEL
LIN {X 0,Y 396.736,Z 513.445,A -85,B 0,C 180,E1 -11271.294,E2 -11271.294} C_VEL
LIN {X 0,Y 397.302,Z 504.597,A -85,B 0,C 180,E1 -11275.122,E2 -11275.122} C_VEL
LIN {X 0,Y 397.902,Z 496.997,A -85,B 0,C 180,E1 -11278.482,E2 -11278.482} C_VEL
LIN {X 0,Y 398.589,Z 488.859,A -85,B 0,C 180,E1 -11282.183,E2 -11282.183} C_VEL
LIN {X 0,Y 399.147,Z 483.024,A -85,B 0,C 180,E1 -11284.907,E2 -11284.907} C_VEL
LIN {X 0,Y 399.21,Z 479.166,A -85,B 0,C 180,E1 -11286.767,E2 -11286.767} C_VEL
LIN {X 0,Y 398.191,Z 472.881,A -85,B 0,C 180,E1 -11290.007,E2 -11290.007} C_VEL
LIN {X 0,Y 397.158,Z 467.015,A -85,B 0,C 180,E1 -11293.215,E2 -11293.215} C_VEL
LIN {X 0,Y 397.165,Z 467.015,A -85,B 0,C 180,E1 -11296.511,E2 -11296.511} C_VEL
LIN {X 0,Y 397.115,Z 467.017,A -85,B 0,C 180,E1 -11299.552,E2 -11299.552} C_VEL
LIN {X 0,Y 397.1,Z 467.021,A -85,B 0,C 180,E1 -11303.005,E2 -11303.005} C_VEL
LIN {X 0,Y 397.119,Z 467.019,A -85,B 0,C 180,E1 -11306.282,E2 -11306.282} C_VEL
LIN {X 0,Y 397.106,Z 467.02,A -85,B 0,C 180,E1 -11310.135,E2 -11310.135} C_VEL
LIN {X 0,Y 397.196,Z 467.01,A -85,B 0,C 180,E1 -11312.61,E2 -11312.61} C_VEL
LIN {X 0,Y 397.134,Z 467.014,A -85,B 0,C 180,E1 -11315.982,E2 -11315.982} C_VEL
LIN {X 0,Y 397.14,Z 467.014,A -85,B 0,C 180,E1 -11319.705,E2 -11319.705} C_VEL
LIN {X 0,Y 397.183,Z 467.011,A -85,B 0,C 180,E1 -11322.845,E2 -11322.845} C_VEL
LIN {X 0,Y 397.23,Z 467.006,A -85,B 0,C 180,E1 -11326.703,E2 -11326.703} C_VEL
LIN {X 0,Y 397.22,Z 467.003,A -85,B 0,C 180,E1 -11329.809,E2 -11329.809} C_VEL
LIN {X 0,Y 397.366,Z 466.989,A -85,B 0,C 180,E1 -11332.888,E2 -11332.888} C_VEL
LIN {X 0,Y 397.256,Z 467.002,A -85,B 0,C 180,E1 -11334.925,E2 -11334.925} C_VEL
LIN {X 0,Y 397.451,Z 466.976,A -85,B 0,C 180,E1 -11337.973,E2 -11337.973} C_VEL
LIN {X 0,Y 397.583,Z 466.961,A -85,B 0,C 180,E1 -11340,E2 -11340} C_VEL
LIN {X 0,Y 397.382,Z 466.985,A -85,B 0,C 180,E1 -11343.042,E2 -11343.042} C_VEL
LIN {X 0,Y 397.366,Z 466.987,A -85,B 0,C 180,E1 -11347.112,E2 -11347.112} C_VEL
LIN {X 0,Y 397.22,Z 467.006,A -85,B 0,C 180,E1 -11350.191,E2 -11350.191} C_VEL
LIN {X 0,Y 397.228,Z 467.003,A -85,B 0,C 180,E1 -11353.321,E2 -11353.321} C_VEL
LIN {X 0,Y 397.184,Z 467.009,A -85,B 0,C 180,E1 -11357.155,E2 -11357.155} C_VEL
LIN {X 0,Y 397.105,Z 467.021,A -85,B 0,C 180,E1 -11360.73,E2 -11360.73} C_VEL
LIN {X 0,Y 397.135,Z 467.017,A -85,B 0,C 180,E1 -11364.018,E2 -11364.018} C_VEL
LIN {X 0,Y 397.197,Z 467.007,A -85,B 0,C 180,E1 -11367.39,E2 -11367.39} C_VEL
LIN {X 0,Y 397.081,Z 467.023,A -85,B 0,C 180,E1 -11370.883,E2 -11370.883} C_VEL
LIN {X 0,Y 397.129,Z 467.018,A -85,B 0,C 180,E1 -11374.493,E2 -11374.493} C_VEL
LIN {X 0,Y 397.106,Z 467.021,A -85,B 0,C 180,E1 -11378.275,E2 -11378.275} C_VEL
LIN {X 0,Y 397.091,Z 467.02,A -85,B 0,C 180,E1 -11380.909,E2 -11380.909} C_VEL
LIN {X 0,Y 397.106,Z 467.02,A -85,B 0,C 180,E1 -11383.648,E2 -11383.648} C_VEL
LIN {X 0,Y 397.106,Z 467.021,A -85,B 0,C 180,E1 -11386.521,E2 -11386.521} C_VEL
LIN {X 0,Y 397.117,Z 467.02,A -85,B 0,C 180,E1 -11390.423,E2 -11390.423} C_VEL
LIN {X 0,Y 397.112,Z 467.022,A -85,B 0,C 180,E1 -11394.266,E2 -11394.266} C_VEL
LIN {X 0,Y 397.118,Z 467.018,A -85,B 0,C 180,E1 -11396.727,E2 -11396.727} C_VEL
LIN {X 0,Y 397.128,Z 467.02,A -85,B 0,C 180,E1 -11400.296,E2 -11400.296} C_VEL
LIN {X 0,Y 397.198,Z 467.008,A -85,B 0,C 180,E1 -11402.61,E2 -11402.61} C_VEL
LIN {X 0,Y 397.137,Z 467.017,A -85,B 0,C 180,E1 -11405.982,E2 -11405.982} C_VEL
LIN {X 0,Y 397.143,Z 467.015,A -85,B 0,C 180,E1 -11409.705,E2 -11409.705} C_VEL
LIN {X 0,Y 397.186,Z 467.009,A -85,B 0,C 180,E1 -11412.845,E2 -11412.845} C_VEL
LIN {X 0,Y 397.233,Z 467.002,A -85,B 0,C 180,E1 -11416.703,E2 -11416.703} C_VEL
LIN {X 0,Y 397.222,Z 467.007,A -85,B 0,C 180,E1 -11419.809,E2 -11419.809} C_VEL
LIN {X 0,Y 397.322,Z 466.991,A -85,B 0,C 180,E1 -11422.888,E2 -11422.888} C_VEL
LIN {X 0,Y 397.253,Z 466.999,A -85,B 0,C 180,E1 -11424.925,E2 -11424.925} C_VEL
LIN {X 0,Y 397.454,Z 466.978,A -85,B 0,C 180,E1 -11427.973,E2 -11427.973} C_VEL
LIN {X 0,Y 397.584,Z 466.963,A -85,B 0,C 180,E1 -11430,E2 -11430} C_VEL
LIN {X 0,Y 397.38,Z 466.984,A -85,B 0,C 180,E1 -11433.042,E2 -11433.042} C_VEL
LIN {X 0,Y 397.373,Z 466.989,A -85,B 0,C 180,E1 -11436.092,E2 -11436.092} C_VEL
LIN {X 0,Y 397.256,Z 466.999,A -85,B 0,C 180,E1 -11439.162,E2 -11439.162} C_VEL
LIN {X 0,Y 397.224,Z 467.007,A -85,B 0,C 180,E1 -11442.258,E2 -11442.258} C_VEL
LIN {X 0,Y 397.184,Z 467.009,A -85,B 0,C 180,E1 -11445.392,E2 -11445.392} C_VEL
LIN {X 0,Y 397.167,Z 467.012,A -85,B 0,C 180,E1 -11448.573,E2 -11448.573} C_VEL
LIN {X 0,Y 397.097,Z 467.022,A -85,B 0,C 180,E1 -11451.91,E2 -11451.91} C_VEL
LIN {X 0,Y 397.157,Z 467.015,A -85,B 0,C 180,E1 -11455.512,E2 -11455.512} C_VEL
LIN {X 0,Y 397.139,Z 467.017,A -85,B 0,C 180,E1 -11456.322,E2 -11456.322} C_VEL
LIN {X 0,Y 396.469,Z 467.1,A -85,B 0,C 180,E1 -11457.168,E2 -11457.168} C_VEL
LIN {X 0,Y 393.594,Z 467.456,A -85,B 0,C 180,E1 -11458.544,E2 -11458.544} C_VEL
LIN {X 0,Y 391.156,Z 467.762,A -85,B 0,C 180,E1 -11459.655,E2 -11459.655} C_VEL
LIN {X 0,Y 390.104,Z 467.89,A -85,B 0,C 180,E1 -11460.515,E2 -11460.515} C_VEL
LIN {X 0,Y 390.016,Z 467.9,A -85,B 0,C 180,E1 -11460.806,E2 -11460.806} C_VEL
LIN {X 0,Y 390.072,Z 467.898,A -85,B 0,C 180,E1 -11464.025,E2 -11464.025} C_VEL
LIN {X 0,Y 390.049,Z 467.9,A -85,B 0,C 180,E1 -11467.551,E2 -11467.551} C_VEL
LIN {X 0,Y 390.06,Z 467.896,A -85,B 0,C 180,E1 -11470.821,E2 -11470.821} C_VEL
LIN {X 0,Y 390.058,Z 467.9,A -85,B 0,C 180,E1 -11473.886,E2 -11473.886} C_VEL
LIN {X 0,Y 390.061,Z 467.896,A -85,B 0,C 180,E1 -11476.79,E2 -11476.79} C_VEL
LIN {X 0,Y 390.06,Z 467.899,A -85,B 0,C 180,E1 -11479.56,E2 -11479.56} C_VEL
LIN {X 0,Y 390.04,Z 467.898,A -85,B 0,C 180,E1 -11482.45,E2 -11482.45} C_VEL
LIN {X 0,Y 389.929,Z 467.912,A -85,B 0,C 180,E1 -11484.776,E2 -11484.776} C_VEL
LIN {X 0,Y 389.556,Z 467.96,A -85,B 0,C 180,E1 -11488.453,E2 -11488.453} C_VEL
LIN {X 0,Y 389.307,Z 467.994,A -85,B 0,C 180,E1 -11490.829,E2 -11490.829} C_VEL
LIN {X 0,Y 389.215,Z 468.579,A -85,B 0,C 180,E1 -11492.226,E2 -11492.226} C_VEL
LIN {X 0,Y 389.074,Z 471.747,A -85,B 0,C 180,E1 -11495.451,E2 -11495.451} C_VEL
LIN {X 0,Y 389.007,Z 475.137,A -85,B 0,C 180,E1 -11498.818,E2 -11498.818} C_VEL
LIN {X 0,Y 388.952,Z 478.569,A -85,B 0,C 180,E1 -11502.144,E2 -11502.144} C_VEL
LIN {X 0,Y 392.368,Z 494.104,A -85,B 0,C 180,E1 -11502.948,E2 -11502.948} C_VEL
LIN {X 0,Y 393.942,Z 502.475,A -85,B 0,C 180,E1 -11503.481,E2 -11503.481} C_VEL
LIN {X 0,Y 393.251,Z 514.547,A -85,B 0,C 180,E1 -11504.317,E2 -11504.317} C_VEL
LIN {X 0,Y 392.562,Z 526.198,A -85,B 0,C 180,E1 -11505.35,E2 -11505.35} C_VEL
LIN {X 0,Y 391.73,Z 537.837,A -85,B 0,C 180,E1 -11506.644,E2 -11506.644} C_VEL
LIN {X 0,Y 391.045,Z 546.392,A -85,B 0,C 180,E1 -11507.809,E2 -11507.809} C_VEL
LIN {X 0,Y 390.376,Z 555.72,A -85,B 0,C 180,E1 -11509.366,E2 -11509.366} C_VEL
LIN {X 0,Y 389.834,Z 563.257,A -85,B 0,C 180,E1 -11510.924,E2 -11510.924} C_VEL
LIN {X 0,Y 389.488,Z 568.386,A -85,B 0,C 180,E1 -11512.222,E2 -11512.222} C_VEL
LIN {X 0,Y 389.249,Z 573.377,A -85,B 0,C 180,E1 -11513.781,E2 -11513.781} C_VEL
LIN {X 0,Y 389.008,Z 577.226,A -85,B 0,C 180,E1 -11515.337,E2 -11515.337} C_VEL
LIN {X 0,Y 388.995,Z 580.02,A -85,B 0,C 180,E1 -11516.893,E2 -11516.893} C_VEL
LIN {X 0,Y 388.901,Z 581.359,A -85,B 0,C 180,E1 -11517.929,E2 -11517.929} C_VEL
LIN {X 0,Y 388.817,Z 582.26,A -85,B 0,C 180,E1 -11518.964,E2 -11518.964} C_VEL
LIN {X 0,Y 388.865,Z 582.813,A -85,B 0,C 180,E1 -11521.035,E2 -11521.035} C_VEL
LIN {X 0,Y 388.95,Z 582.499,A -85,B 0,C 180,E1 -11522.071,E2 -11522.071} C_VEL
LIN {X 0,Y 389.06,Z 581.74,A -85,B 0,C 180,E1 -11523.106,E2 -11523.106} C_VEL
LIN {X 0,Y 389.233,Z 580.566,A -85,B 0,C 180,E1 -11524.142,E2 -11524.142} C_VEL
LIN {X 0,Y 389.265,Z 578.047,A -85,B 0,C 180,E1 -11525.699,E2 -11525.699} C_VEL
LIN {X 0,Y 389.76,Z 574.17,A -85,B 0,C 180,E1 -11527.368,E2 -11527.368} C_VEL
LIN {X 0,Y 390.194,Z 569.816,A -85,B 0,C 180,E1 -11528.806,E2 -11528.806} C_VEL
LIN {X 0,Y 390.889,Z 563.945,A -85,B 0,C 180,E1 -11530.358,E2 -11530.358} C_VEL
LIN {X 0,Y 391.624,Z 556.676,A -85,B 0,C 180,E1 -11531.91,E2 -11531.91} C_VEL
LIN {X 0,Y 392.5,Z 547.6,A -85,B 0,C 180,E1 -11533.46,E2 -11533.46} C_VEL
LIN {X 0,Y 393.701,Z 538.377,A -85,B 0,C 180,E1 -11534.724,E2 -11534.724} C_VEL
LIN {X 0,Y 394.751,Z 527.388,A -85,B 0,C 180,E1 -11535.971,E2 -11535.971} C_VEL
LIN {X 0,Y 395.842,Z 515.603,A -85,B 0,C 180,E1 -11537.035,E2 -11537.035} C_VEL
LIN {X 0,Y 396.564,Z 505.609,A -85,B 0,C 180,E1 -11537.764,E2 -11537.764} C_VEL
LIN {X 0,Y 394.524,Z 497.233,A -85,B 0,C 180,E1 -11538.451,E2 -11538.451} C_VEL
LIN {X 0,Y 390.745,Z 486.365,A -85,B 0,C 180,E1 -11539.321,E2 -11539.321} C_VEL
LIN {X 0,Y 389.72,Z 483.389,A -85,B 0,C 180,E1 -11539.557,E2 -11539.557} C_VEL
LIN {X 0,Y 389.899,Z 480.866,A -85,B 0,C 180,E1 -11543.363,E2 -11543.363} C_VEL
LIN {X 0,Y 390.162,Z 478.9,A -85,B 0,C 180,E1 -11546.765,E2 -11546.765} C_VEL
LIN {X 0,Y 390.384,Z 477.752,A -85,B 0,C 180,E1 -11549.083,E2 -11549.083} C_VEL
LIN {X 0,Y 390.805,Z 476.394,A -85,B 0,C 180,E1 -11552.65,E2 -11552.65} C_VEL
LIN {X 0,Y 391.058,Z 475.774,A -85,B 0,C 180,E1 -11555.106,E2 -11555.106} C_VEL
LIN {X 0,Y 391.287,Z 475.485,A -85,B 0,C 180,E1 -11557.786,E2 -11557.786} C_VEL
LIN {X 0,Y 391.421,Z 475.813,A -85,B 0,C 180,E1 -11561.052,E2 -11561.052} C_VEL
LIN {X 0,Y 391.682,Z 476.982,A -85,B 0,C 180,E1 -11564.41,E2 -11564.41} C_VEL
LIN {X 0,Y 392.015,Z 478.75,A -85,B 0,C 180,E1 -11567.311,E2 -11567.311} C_VEL
LIN {X 0,Y 392.407,Z 481.41,A -85,B 0,C 180,E1 -11570.366,E2 -11570.366} C_VEL
LIN {X 0,Y 392.699,Z 483.805,A -85,B 0,C 180,E1 -11572.52,E2 -11572.52} C_VEL
LIN {X 0,Y 392.457,Z 487.241,A -85,B 0,C 180,E1 -11575.037,E2 -11575.037} C_VEL
LIN {X 0,Y 391.706,Z 492.077,A -85,B 0,C 180,E1 -11578.042,E2 -11578.042} C_VEL
LIN {X 0,Y 390.972,Z 497.333,A -85,B 0,C 180,E1 -11580.965,E2 -11580.965} C_VEL
LIN {X 0,Y 390.324,Z 504.131,A -85,B 0,C 180,E1 -11584.397,E2 -11584.397} C_VEL
LIN {X 0,Y 389.702,Z 512.504,A -85,B 0,C 180,E1 -11588.302,E2 -11588.302} C_VEL
LIN {X 0,Y 389.446,Z 517.406,A -85,B 0,C 180,E1 -11590.394,E2 -11590.394} C_VEL
LIN {X 0,Y 392.384,Z 530.708,A -85,B 0,C 180,E1 -11591.192,E2 -11591.192} C_VEL
LIN {X 0,Y 393.928,Z 542.735,A -85,B 0,C 180,E1 -11591.989,E2 -11591.989} C_VEL
LIN {X 0,Y 394.373,Z 556.404,A -85,B 0,C 180,E1 -11593.033,E2 -11593.033} C_VEL
LIN {X 0,Y 393.294,Z 568.064,A -85,B 0,C 180,E1 -11594.053,E2 -11594.053} C_VEL
LIN {X 0,Y 392.102,Z 579.777,A -85,B 0,C 180,E1 -11595.334,E2 -11595.334} C_VEL
LIN {X 0,Y 391.015,Z 590.32,A -85,B 0,C 180,E1 -11596.752,E2 -11596.752} C_VEL
LIN {X 0,Y 390.196,Z 599.62,A -85,B 0,C 180,E1 -11598.309,E2 -11598.309} C_VEL
LIN {X 0,Y 389.548,Z 607.232,A -85,B 0,C 180,E1 -11599.869,E2 -11599.869} C_VEL
LIN {X 0,Y 389.106,Z 614.315,A -85,B 0,C 180,E1 -11601.692,E2 -11601.692} C_VEL
LIN {X 0,Y 388.882,Z 619.045,A -85,B 0,C 180,E1 -11603.254,E2 -11603.254} C_VEL
LIN {X 0,Y 388.769,Z 622.674,A -85,B 0,C 180,E1 -11604.814,E2 -11604.814} C_VEL
LIN {X 0,Y 388.739,Z 624.504,A -85,B 0,C 180,E1 -11605.853,E2 -11605.853} C_VEL
LIN {X 0,Y 388.743,Z 625.915,A -85,B 0,C 180,E1 -11606.891,E2 -11606.891} C_VEL
LIN {X 0,Y 388.845,Z 626.911,A -85,B 0,C 180,E1 -11607.928,E2 -11607.928} C_VEL
LIN {X 0,Y 388.801,Z 627.435,A -85,B 0,C 180,E1 -11608.964,E2 -11608.964} C_VEL
LIN {X 0,Y 388.81,Z 627.549,A -85,B 0,C 180,E1 -11610,E2 -11610} C_VEL
LIN {X 0,Y 388.81,Z 627.253,A -85,B 0,C 180,E1 -11611.036,E2 -11611.036} C_VEL
LIN {X 0,Y 388.848,Z 626.531,A -85,B 0,C 180,E1 -11612.071,E2 -11612.071} C_VEL
LIN {X 0,Y 388.78,Z 625.336,A -85,B 0,C 180,E1 -11613.109,E2 -11613.109} C_VEL
LIN {X 0,Y 388.813,Z 622.746,A -85,B 0,C 180,E1 -11614.665,E2 -11614.665} C_VEL
LIN {X 0,Y 388.834,Z 619.083,A -85,B 0,C 180,E1 -11616.226,E2 -11616.226} C_VEL
LIN {X 0,Y 389.01,Z 614.268,A -85,B 0,C 180,E1 -11617.787,E2 -11617.787} C_VEL
LIN {X 0,Y 389.31,Z 608.16,A -85,B 0,C 180,E1 -11619.35,E2 -11619.35} C_VEL
LIN {X 0,Y 389.749,Z 600.554,A -85,B 0,C 180,E1 -11620.914,E2 -11620.914} C_VEL
LIN {X 0,Y 390.369,Z 592.811,A -85,B 0,C 180,E1 -11622.213,E2 -11622.213} C_VEL
LIN {X 0,Y 391.023,Z 583.389,A -85,B 0,C 180,E1 -11623.512,E2 -11623.512} C_VEL
LIN {X 0,Y 391.879,Z 571.798,A -85,B 0,C 180,E1 -11624.807,E2 -11624.807} C_VEL
LIN {X 0,Y 392.678,Z 560.102,A -85,B 0,C 180,E1 -11625.839,E2 -11625.839} C_VEL
LIN {X 0,Y 393.159,Z 553.045,A -85,B 0,C 180,E1 -11626.352,E2 -11626.352} C_VEL
LIN {X 0,Y 391.93,Z 541.269,A -85,B 0,C 180,E1 -11627.11,E2 -11627.11} C_VEL
LIN {X 0,Y 390.051,Z 527.093,A -85,B 0,C 180,E1 -11627.798,E2 -11627.798} C_VEL
LIN {X 0,Y 389.306,Z 521.34,A -85,B 0,C 180,E1 -11628.042,E2 -11628.042} C_VEL
LIN {X 0,Y 389.704,Z 512.956,A -85,B 0,C 180,E1 -11631.697,E2 -11631.697} C_VEL
LIN {X 0,Y 390.217,Z 505.397,A -85,B 0,C 180,E1 -11635.04,E2 -11635.04} C_VEL
LIN {X 0,Y 390.81,Z 498.371,A -85,B 0,C 180,E1 -11638.215,E2 -11638.215} C_VEL
LIN {X 0,Y 391.489,Z 490.314,A -85,B 0,C 180,E1 -11641.938,E2 -11641.938} C_VEL
LIN {X 0,Y 392.138,Z 483.882,A -85,B 0,C 180,E1 -11644.995,E2 -11644.995} C_VEL
LIN {X 0,Y 392.165,Z 480.044,A -85,B 0,C 180,E1 -11646.895,E2 -11646.895} C_VEL
LIN {X 0,Y 391.397,Z 475.121,A -85,B 0,C 180,E1 -11649.456,E2 -11649.456} C_VEL
LIN {X 0,Y 390.161,Z 468.126,A -85,B 0,C 180,E1 -11653.293,E2 -11653.293} C_VEL
LIN {X 0,Y 390.066,Z 467.898,A -85,B 0,C 180,E1 -11653.888,E2 -11653.888} C_VEL
LIN {X 0,Y 390.118,Z 467.892,A -85,B 0,C 180,E1 -11656.798,E2 -11656.798} C_VEL
LIN {X 0,Y 390.07,Z 467.894,A -85,B 0,C 180,E1 -11659.562,E2 -11659.562} C_VEL
LIN {X 0,Y 390.043,Z 467.901,A -85,B 0,C 180,E1 -11662.449,E2 -11662.449} C_VEL
LIN {X 0,Y 390.069,Z 467.895,A -85,B 0,C 180,E1 -11665.975,E2 -11665.975} C_VEL
LIN {X 0,Y 390.048,Z 467.897,A -85,B 0,C 180,E1 -11669.869,E2 -11669.869} C_VEL
LIN {X 0,Y 390.115,Z 467.89,A -85,B 0,C 180,E1 -11673.232,E2 -11673.232} C_VEL
LIN {X 0,Y 390.108,Z 467.893,A -85,B 0,C 180,E1 -11676.75,E2 -11676.75} C_VEL
LIN {X 0,Y 390.105,Z 467.891,A -85,B 0,C 180,E1 -11679.983,E2 -11679.983} C_VEL
LIN {X 0,Y 390.14,Z 467.886,A -85,B 0,C 180,E1 -11683.248,E2 -11683.248} C_VEL
LIN {X 0,Y 390.196,Z 467.882,A -85,B 0,C 180,E1 -11686.562,E2 -11686.562} C_VEL
LIN {X 0,Y 390.17,Z 467.881,A -85,B 0,C 180,E1 -11689.623,E2 -11689.623} C_VEL
LIN {X 0,Y 390.32,Z 467.866,A -85,B 0,C 180,E1 -11692.759,E2 -11692.759} C_VEL
LIN {X 0,Y 390.228,Z 467.878,A -85,B 0,C 180,E1 -11694.834,E2 -11694.834} C_VEL
LIN {X 0,Y 390.42,Z 467.851,A -85,B 0,C 180,E1 -11697.937,E2 -11697.937} C_VEL
LIN {X 0,Y 390.552,Z 467.836,A -85,B 0,C 180,E1 -11700,E2 -11700} C_VEL
LIN {X 0,Y 390.316,Z 467.864,A -85,B 0,C 180,E1 -11703.097,E2 -11703.097} C_VEL
LIN {X 0,Y 390.312,Z 467.865,A -85,B 0,C 180,E1 -11706.642,E2 -11706.642} C_VEL
LIN {X 0,Y 390.207,Z 467.878,A -85,B 0,C 180,E1 -11709.329,E2 -11709.329} C_VEL
LIN {X 0,Y 390.196,Z 467.879,A -85,B 0,C 180,E1 -11713.439,E2 -11713.439} C_VEL
LIN {X 0,Y 390.151,Z 467.884,A -85,B 0,C 180,E1 -11717.308,E2 -11717.308} C_VEL
LIN {X 0,Y 390.089,Z 467.895,A -85,B 0,C 180,E1 -11720.47,E2 -11720.47} C_VEL
LIN {X 0,Y 390.092,Z 467.892,A -85,B 0,C 180,E1 -11723.351,E2 -11723.351} C_VEL
LIN {X 0,Y 390.116,Z 467.89,A -85,B 0,C 180,E1 -11726.768,E2 -11726.768} C_VEL
LIN {X 0,Y 390.041,Z 467.901,A -85,B 0,C 180,E1 -11730.3,E2 -11730.3} C_VEL
LIN {X 0,Y 390.071,Z 467.897,A -85,B 0,C 180,E1 -11734.025,E2 -11734.025} C_VEL
LIN {X 0,Y 390.047,Z 467.898,A -85,B 0,C 180,E1 -11737.551,E2 -11737.551} C_VEL
LIN {X 0,Y 390.059,Z 467.897,A -85,B 0,C 180,E1 -11740.822,E2 -11740.822} C_VEL
LIN {X 0,Y 390.06,Z 467.899,A -85,B 0,C 180,E1 -11743.887,E2 -11743.887} C_VEL
LIN {X 0,Y 390.061,Z 467.896,A -85,B 0,C 180,E1 -11746.79,E2 -11746.79} C_VEL
LIN {X 0,Y 390.059,Z 467.896,A -85,B 0,C 180,E1 -11749.561,E2 -11749.561} C_VEL
LIN {X 0,Y 390.049,Z 467.901,A -85,B 0,C 180,E1 -11752.449,E2 -11752.449} C_VEL
LIN {X 0,Y 390.087,Z 467.897,A -85,B 0,C 180,E1 -11756.047,E2 -11756.047} C_VEL
LIN {X 0,Y 390.05,Z 467.9,A -85,B 0,C 180,E1 -11759.869,E2 -11759.869} C_VEL
LIN {X 0,Y 390.117,Z 467.888,A -85,B 0,C 180,E1 -11763.232,E2 -11763.232} C_VEL
LIN {X 0,Y 390.11,Z 467.891,A -85,B 0,C 180,E1 -11766.75,E2 -11766.75} C_VEL
LIN {X 0,Y 390.108,Z 467.894,A -85,B 0,C 180,E1 -11769.983,E2 -11769.983} C_VEL
LIN {X 0,Y 390.142,Z 467.886,A -85,B 0,C 180,E1 -11773.248,E2 -11773.248} C_VEL
LIN {X 0,Y 390.199,Z 467.879,A -85,B 0,C 180,E1 -11776.562,E2 -11776.562} C_VEL
LIN {X 0,Y 390.208,Z 467.879,A -85,B 0,C 180,E1 -11780.671,E2 -11780.671} C_VEL
LIN {X 0,Y 390.313,Z 467.867,A -85,B 0,C 180,E1 -11783.798,E2 -11783.798} C_VEL
LIN {X 0,Y 390.423,Z 467.854,A -85,B 0,C 180,E1 -11787.937,E2 -11787.937} C_VEL
LIN {X 0,Y 390.553,Z 467.838,A -85,B 0,C 180,E1 -11790,E2 -11790} C_VEL
LIN {X 0,Y 390.315,Z 467.864,A -85,B 0,C 180,E1 -11793.097,E2 -11793.097} C_VEL
LIN {X 0,Y 390.326,Z 467.867,A -85,B 0,C 180,E1 -11796.202,E2 -11796.202} C_VEL
LIN {X 0,Y 390.208,Z 467.878,A -85,B 0,C 180,E1 -11799.329,E2 -11799.329} C_VEL
LIN {X 0,Y 390.176,Z 467.883,A -85,B 0,C 180,E1 -11802.483,E2 -11802.483} C_VEL
LIN {X 0,Y 390.144,Z 467.888,A -85,B 0,C 180,E1 -11805.677,E2 -11805.677} C_VEL
LIN {X 0,Y 390.11,Z 467.89,A -85,B 0,C 180,E1 -11808.922,E2 -11808.922} C_VEL
LIN {X 0,Y 390.045,Z 467.899,A -85,B 0,C 180,E1 -11812.234,E2 -11812.234} C_VEL
LIN {X 0,Y 390.124,Z 467.891,A -85,B 0,C 180,E1 -11815.743,E2 -11815.743} C_VEL
LIN {X 0,Y 390.062,Z 467.896,A -85,B 0,C 180,E1 -11819.109,E2 -11819.109} C_VEL
LIN {X 0,Y 390.016,Z 467.9,A -85,B 0,C 180,E1 -11820.806,E2 -11820.806} C_VEL
LIN {X 0,Y 389.342,Z 467.99,A -85,B 0,C 180,E1 -11821.668,E2 -11821.668} C_VEL
LIN {X 0,Y 386.495,Z 468.34,A -85,B 0,C 180,E1 -11823.07,E2 -11823.07} C_VEL
LIN {X 0,Y 384.097,Z 468.641,A -85,B 0,C 180,E1 -11824.203,E2 -11824.203} C_VEL
LIN {X 0,Y 383.079,Z 468.766,A -85,B 0,C 180,E1 -11825.079,E2 -11825.079} C_VEL
LIN {X 0,Y 383.002,Z 468.774,A -85,B 0,C 180,E1 -11825.375,E2 -11825.375} C_VEL
LIN {X 0,Y 383.009,Z 468.774,A -85,B 0,C 180,E1 -11828.6,E2 -11828.6} C_VEL
LIN {X 0,Y 382.988,Z 468.779,A -85,B 0,C 180,E1 -11831.347,E2 -11831.347} C_VEL
LIN {X 0,Y 382.999,Z 468.776,A -85,B 0,C 180,E1 -11834.303,E2 -11834.303} C_VEL
LIN {X 0,Y 383.013,Z 468.775,A -85,B 0,C 180,E1 -11837.24,E2 -11837.24} C_VEL
LIN {X 0,Y 383.018,Z 468.773,A -85,B 0,C 180,E1 -11840.413,E2 -11840.413} C_VEL
LIN {X 0,Y 382.944,Z 468.785,A -85,B 0,C 180,E1 -11843.854,E2 -11843.854} C_VEL
LIN {X 0,Y 382.693,Z 468.814,A -85,B 0,C 180,E1 -11846.568,E2 -11846.568} C_VEL
LIN {X 0,Y 382.345,Z 468.862,A -85,B 0,C 180,E1 -11850.244,E2 -11850.244} C_VEL
LIN {X 0,Y 382.177,Z 469.015,A -85,B 0,C 180,E1 -11851.969,E2 -11851.969} C_VEL
LIN {X 0,Y 382.043,Z 471.923,A -85,B 0,C 180,E1 -11854.969,E2 -11854.969} C_VEL
LIN {X 0,Y 381.949,Z 475.351,A -85,B 0,C 180,E1 -11858.407,E2 -11858.407} C_VEL
LIN {X 0,Y 381.922,Z 478.944,A -85,B 0,C 180,E1 -11861.916,E2 -11861.916} C_VEL
LIN {X 0,Y 385.103,Z 493.829,A -85,B 0,C 180,E1 -11862.673,E2 -11862.673} C_VEL
LIN {X 0,Y 387.008,Z 503.618,A -85,B 0,C 180,E1 -11863.312,E2 -11863.312} C_VEL
LIN {X 0,Y 386.278,Z 515.521,A -85,B 0,C 180,E1 -11864.162,E2 -11864.162} C_VEL
LIN {X 0,Y 385.56,Z 527.034,A -85,B 0,C 180,E1 -11865.215,E2 -11865.215} C_VEL
LIN {X 0,Y 384.711,Z 538.569,A -85,B 0,C 180,E1 -11866.531,E2 -11866.531} C_VEL
LIN {X 0,Y 383.964,Z 547.901,A -85,B 0,C 180,E1 -11867.848,E2 -11867.848} C_VEL
LIN {X 0,Y 383.27,Z 557.011,A -85,B 0,C 180,E1 -11869.434,E2 -11869.434} C_VEL
LIN {X 0,Y 382.732,Z 564.394,A -85,B 0,C 180,E1 -11871.02,E2 -11871.02} C_VEL
LIN {X 0,Y 382.376,Z 570.299,A -85,B 0,C 180,E1 -11872.608,E2 -11872.608} C_VEL
LIN {X 0,Y 382.095,Z 574.961,A -85,B 0,C 180,E1 -11874.194,E2 -11874.194} C_VEL
LIN {X 0,Y 381.883,Z 578.521,A -85,B 0,C 180,E1 -11875.778,E2 -11875.778} C_VEL
LIN {X 0,Y 381.901,Z 580.302,A -85,B 0,C 180,E1 -11876.835,E2 -11876.835} C_VEL
LIN {X 0,Y 381.837,Z 581.68,A -85,B 0,C 180,E1 -11877.89,E2 -11877.89} C_VEL
LIN {X 0,Y 381.747,Z 582.645,A -85,B 0,C 180,E1 -11878.945,E2 -11878.945} C_VEL
LIN {X 0,Y 381.727,Z 583.156,A -85,B 0,C 180,E1 -11880,E2 -11880} C_VEL
LIN {X 0,Y 381.793,Z 583.269,A -85,B 0,C 180,E1 -11881.055,E2 -11881.055} C_VEL
LIN {X 0,Y 381.884,Z 582.989,A -85,B 0,C 180,E1 -11882.109,E2 -11882.109} C_VEL
LIN {X 0,Y 382.008,Z 582.285,A -85,B 0,C 180,E1 -11883.164,E2 -11883.164} C_VEL
LIN {X 0,Y 382.19,Z 581.141,A -85,B 0,C 180,E1 -11884.218,E2 -11884.218} C_VEL
LIN {X 0,Y 382.229,Z 579.612,A -85,B 0,C 180,E1 -11885.275,E2 -11885.275} C_VEL
LIN {X 0,Y 382.605,Z 576.291,A -85,B 0,C 180,E1 -11886.943,E2 -11886.943} C_VEL
LIN {X 0,Y 383.066,Z 572.296,A -85,B 0,C 180,E1 -11888.44,E2 -11888.44} C_VEL
LIN {X 0,Y 383.67,Z 566.944,A -85,B 0,C 180,E1 -11890.021,E2 -11890.021} C_VEL
LIN {X 0,Y 384.44,Z 560.258,A -85,B 0,C 180,E1 -11891.601,E2 -11891.601} C_VEL
LIN {X 0,Y 385.472,Z 551.922,A -85,B 0,C 180,E1 -11893.174,E2 -11893.174} C_VEL
LIN {X 0,Y 386.264,Z 545.359,A -85,B 0,C 180,E1 -11894.219,E2 -11894.219} C_VEL
LIN {X 0,Y 387.483,Z 535.526,A -85,B 0,C 180,E1 -11895.517,E2 -11895.517} C_VEL
LIN {X 0,Y 388.551,Z 524.654,A -85,B 0,C 180,E1 -11896.699,E2 -11896.699} C_VEL
LIN {X 0,Y 389.682,Z 512.747,A -85,B 0,C 180,E1 -11897.719,E2 -11897.719} C_VEL
LIN {X 0,Y 390.068,Z 507.124,A -85,B 0,C 180,E1 -11898.132,E2 -11898.132} C_VEL
LIN {X 0,Y 387.673,Z 497.711,A -85,B 0,C 180,E1 -11898.965,E2 -11898.965} C_VEL
LIN {X 0,Y 383.739,Z 487.004,A -85,B 0,C 180,E1 -11899.879,E2 -11899.879} C_VEL
LIN {X 0,Y 382.709,Z 484.063,A -85,B 0,C 180,E1 -11900.141,E2 -11900.141} C_VEL
LIN {X 0,Y 382.929,Z 481.74,A -85,B 0,C 180,E1 -11903.814,E2 -11903.814} C_VEL
LIN {X 0,Y 383.222,Z 479.872,A -85,B 0,C 180,E1 -11907.289,E2 -11907.289} C_VEL
LIN {X 0,Y 383.617,Z 478.327,A -85,B 0,C 180,E1 -11910.862,E2 -11910.862} C_VEL
LIN {X 0,Y 383.923,Z 477.566,A -85,B 0,C 180,E1 -11913.31,E2 -11913.31} C_VEL
LIN {X 0,Y 384.256,Z 477.034,A -85,B 0,C 180,E1 -11916.413,E2 -11916.413} C_VEL
LIN {X 0,Y 384.432,Z 477.101,A -85,B 0,C 180,E1 -11919.781,E2 -11919.781} C_VEL
LIN {X 0,Y 384.632,Z 477.949,A -85,B 0,C 180,E1 -11923.039,E2 -11923.039} C_VEL
LIN {X 0,Y 384.908,Z 479.462,A -85,B 0,C 180,E1 -11926.065,E2 -11926.065} C_VEL
LIN {X 0,Y 385.276,Z 481.616,A -85,B 0,C 180,E1 -11928.952,E2 -11928.952} C_VEL
LIN {X 0,Y 385.698,Z 484.346,A -85,B 0,C 180,E1 -11931.718,E2 -11931.718} C_VEL
LIN {X 0,Y 385.724,Z 486.243,A -85,B 0,C 180,E1 -11933.292,E2 -11933.292} C_VEL
LIN {X 0,Y 385.393,Z 489.432,A -85,B 0,C 180,E1 -11935.576,E2 -11935.576} C_VEL
LIN {X 0,Y 384.546,Z 494.313,A -85,B 0,C 180,E1 -11938.609,E2 -11938.609} C_VEL
LIN {X 0,Y 383.698,Z 500.738,A -85,B 0,C 180,E1 -11942.155,E2 -11942.155} C_VEL
LIN {X 0,Y 383.029,Z 507.608,A -85,B 0,C 180,E1 -11945.616,E2 -11945.616} C_VEL
LIN {X 0,Y 382.571,Z 514.829,A -85,B 0,C 180,E1 -11949.009,E2 -11949.009} C_VEL
LIN {X 0,Y 382.463,Z 516.581,A -85,B 0,C 180,E1 -11949.808,E2 -11949.808} C_VEL
LIN {X 0,Y 385.644,Z 530.678,A -85,B 0,C 180,E1 -11950.712,E2 -11950.712} C_VEL
LIN {X 0,Y 387.194,Z 542.065,A -85,B 0,C 180,E1 -11951.512,E2 -11951.512} C_VEL
LIN {X 0,Y 387.764,Z 555.766,A -85,B 0,C 180,E1 -11952.599,E2 -11952.599} C_VEL
LIN {X 0,Y 386.647,Z 567.364,A -85,B 0,C 180,E1 -11953.636,E2 -11953.636} C_VEL
LIN {X 0,Y 385.335,Z 579.065,A -85,B 0,C 180,E1 -11954.936,E2 -11954.936} C_VEL
LIN {X 0,Y 384.245,Z 588.714,A -85,B 0,C 180,E1 -11956.245,E2 -11956.245} C_VEL
LIN {X 0,Y 383.559,Z 596.776,A -85,B 0,C 180,E1 -11957.567,E2 -11957.567} C_VEL
LIN {X 0,Y 382.701,Z 604.82,A -85,B 0,C 180,E1 -11959.15,E2 -11959.15} C_VEL
LIN {X 0,Y 382.172,Z 612.295,A -85,B 0,C 180,E1 -11961.007,E2 -11961.007} C_VEL
LIN {X 0,Y 381.855,Z 617.358,A -85,B 0,C 180,E1 -11962.598,E2 -11962.598} C_VEL
LIN {X 0,Y 381.754,Z 620.415,A -85,B 0,C 180,E1 -11963.788,E2 -11963.788} C_VEL
LIN {X 0,Y 381.662,Z 624.172,A -85,B 0,C 180,E1 -11965.776,E2 -11965.776} C_VEL
LIN {X 0,Y 381.646,Z 625.562,A -85,B 0,C 180,E1 -11966.833,E2 -11966.833} C_VEL
LIN {X 0,Y 381.756,Z 626.513,A -85,B 0,C 180,E1 -11967.89,E2 -11967.89} C_VEL
LIN {X 0,Y 381.731,Z 627.011,A -85,B 0,C 180,E1 -11968.945,E2 -11968.945} C_VEL
LIN {X 0,Y 381.736,Z 627.103,A -85,B 0,C 180,E1 -11970,E2 -11970} C_VEL
LIN {X 0,Y 381.739,Z 626.785,A -85,B 0,C 180,E1 -11971.055,E2 -11971.055} C_VEL
LIN {X 0,Y 381.779,Z 626.013,A -85,B 0,C 180,E1 -11972.11,E2 -11972.11} C_VEL
LIN {X 0,Y 381.688,Z 624.792,A -85,B 0,C 180,E1 -11973.166,E2 -11973.166} C_VEL
LIN {X 0,Y 381.746,Z 622.147,A -85,B 0,C 180,E1 -11974.752,E2 -11974.752} C_VEL
LIN {X 0,Y 381.767,Z 618.421,A -85,B 0,C 180,E1 -11976.341,E2 -11976.341} C_VEL
LIN {X 0,Y 381.934,Z 613.534,A -85,B 0,C 180,E1 -11977.933,E2 -11977.933} C_VEL
LIN {X 0,Y 382.238,Z 607.349,A -85,B 0,C 180,E1 -11979.525,E2 -11979.525} C_VEL
LIN {X 0,Y 382.715,Z 599.646,A -85,B 0,C 180,E1 -11981.117,E2 -11981.117} C_VEL
LIN {X 0,Y 383.428,Z 590.003,A -85,B 0,C 180,E1 -11982.706,E2 -11982.706} C_VEL
LIN {X 0,Y 384.169,Z 580.129,A -85,B 0,C 180,E1 -11984.028,E2 -11984.028} C_VEL
LIN {X 0,Y 385.049,Z 569.124,A -85,B 0,C 180,E1 -11985.211,E2 -11985.211} C_VEL
LIN {X 0,Y 385.945,Z 556.916,A -85,B 0,C 180,E1 -11986.259,E2 -11986.259} C_VEL
LIN {X 0,Y 385.923,Z 551.329,A -85,B 0,C 180,E1 -11986.668,E2 -11986.668} C_VEL
LIN {X 0,Y 384.475,Z 538.378,A -85,B 0,C 180,E1 -11987.481,E2 -11987.481} C_VEL
LIN {X 0,Y 382.651,Z 524.459,A -85,B 0,C 180,E1 -11988.141,E2 -11988.141} C_VEL
LIN {X 0,Y 382.243,Z 521.05,A -85,B 0,C 180,E1 -11988.283,E2 -11988.283} C_VEL
LIN {X 0,Y 382.682,Z 512.464,A -85,B 0,C 180,E1 -11992.116,E2 -11992.116} C_VEL
LIN {X 0,Y 383.316,Z 503.799,A -85,B 0,C 180,E1 -11996.051,E2 -11996.051} C_VEL
LIN {X 0,Y 383.891,Z 497.381,A -85,B 0,C 180,E1 -11999.021,E2 -11999.021} C_VEL
LIN {X 0,Y 384.658,Z 489.4,A -85,B 0,C 180,E1 -12002.812,E2 -12002.812} C_VEL
LIN {X 0,Y 385.21,Z 483.451,A -85,B 0,C 180,E1 -12005.72,E2 -12005.72} C_VEL
LIN {X 0,Y 384.969,Z 479.718,A -85,B 0,C 180,E1 -12007.627,E2 -12007.627} C_VEL
LIN {X 0,Y 384.051,Z 474.374,A -85,B 0,C 180,E1 -12010.514,E2 -12010.514} C_VEL
LIN {X 0,Y 383.033,Z 468.774,A -85,B 0,C 180,E1 -12013.738,E2 -12013.738} C_VEL
LIN {X 0,Y 383.076,Z 468.768,A -85,B 0,C 180,E1 -12017.249,E2 -12017.249} C_VEL
LIN {X 0,Y 383.018,Z 468.775,A -85,B 0,C 180,E1 -12020.413,E2 -12020.413} C_VEL
LIN {X 0,Y 383.026,Z 468.773,A -85,B 0,C 180,E1 -12024.045,E2 -12024.045} C_VEL
LIN {X 0,Y 382.988,Z 468.776,A -85,B 0,C 180,E1 -12027.578,E2 -12027.578} C_VEL
LIN {X 0,Y 382.993,Z 468.778,A -85,B 0,C 180,E1 -12030.3,E2 -12030.3} C_VEL
LIN {X 0,Y 383.081,Z 468.766,A -85,B 0,C 180,E1 -12034.021,E2 -12034.021} C_VEL
LIN {X 0,Y 383.01,Z 468.774,A -85,B 0,C 180,E1 -12037.335,E2 -12037.335} C_VEL
LIN {X 0,Y 383.062,Z 468.772,A -85,B 0,C 180,E1 -12040.716,E2 -12040.716} C_VEL
LIN {X 0,Y 383.082,Z 468.766,A -85,B 0,C 180,E1 -12044.027,E2 -12044.027} C_VEL
LIN {X 0,Y 383.138,Z 468.758,A -85,B 0,C 180,E1 -12047.284,E2 -12047.284} C_VEL
LIN {X 0,Y 383.153,Z 468.761,A -85,B 0,C 180,E1 -12050.498,E2 -12050.498} C_VEL
LIN {X 0,Y 383.275,Z 468.744,A -85,B 0,C 180,E1 -12052.625,E2 -12052.625} C_VEL
LIN {X 0,Y 383.2,Z 468.754,A -85,B 0,C 180,E1 -12054.739,E2 -12054.739} C_VEL
LIN {X 0,Y 383.387,Z 468.727,A -85,B 0,C 180,E1 -12057.899,E2 -12057.899} C_VEL
LIN {X 0,Y 383.522,Z 468.712,A -85,B 0,C 180,E1 -12060,E2 -12060} C_VEL
LIN {X 0,Y 383.252,Z 468.744,A -85,B 0,C 180,E1 -12063.154,E2 -12063.154} C_VEL
LIN {X 0,Y 383.271,Z 468.743,A -85,B 0,C 180,E1 -12066.637,E2 -12066.637} C_VEL
LIN {X 0,Y 383.262,Z 468.746,A -85,B 0,C 180,E1 -12068.436,E2 -12068.436} C_VEL
LIN {X 0,Y 383.1,Z 468.762,A -85,B 0,C 180,E1 -12071.642,E2 -12071.642} C_VEL
LIN {X 0,Y 383.112,Z 468.763,A -85,B 0,C 180,E1 -12074.882,E2 -12074.882} C_VEL
LIN {X 0,Y 383.091,Z 468.766,A -85,B 0,C 180,E1 -12078.172,E2 -12078.172} C_VEL
LIN {X 0,Y 382.995,Z 468.776,A -85,B 0,C 180,E1 -12081.531,E2 -12081.531} C_VEL
LIN {X 0,Y 383.055,Z 468.769,A -85,B 0,C 180,E1 -12084.96,E2 -12084.96} C_VEL
LIN {X 0,Y 383.042,Z 468.773,A -85,B 0,C 180,E1 -12088.493,E2 -12088.493} C_VEL
LIN {X 0,Y 383.012,Z 468.777,A -85,B 0,C 180,E1 -12092.15,E2 -12092.15} C_VEL
LIN {X 0,Y 383.021,Z 468.775,A -85,B 0,C 180,E1 -12094.668,E2 -12094.668} C_VEL
LIN {X 0,Y 383.003,Z 468.778,A -85,B 0,C 180,E1 -12097.904,E2 -12097.904} C_VEL
LIN {X 0,Y 382.987,Z 468.776,A -85,B 0,C 180,E1 -12101.347,E2 -12101.347} C_VEL
LIN {X 0,Y 383.001,Z 468.779,A -85,B 0,C 180,E1 -12104.304,E2 -12104.304} C_VEL
LIN {X 0,Y 383.012,Z 468.773,A -85,B 0,C 180,E1 -12107.24,E2 -12107.24} C_VEL
LIN {X 0,Y 383.019,Z 468.776,A -85,B 0,C 180,E1 -12110.414,E2 -12110.414} C_VEL
LIN {X 0,Y 383.03,Z 468.775,A -85,B 0,C 180,E1 -12114.045,E2 -12114.045} C_VEL
LIN {X 0,Y 382.99,Z 468.777,A -85,B 0,C 180,E1 -12117.578,E2 -12117.578} C_VEL
LIN {X 0,Y 382.996,Z 468.78,A -85,B 0,C 180,E1 -12120.3,E2 -12120.3} C_VEL
LIN {X 0,Y 383.084,Z 468.769,A -85,B 0,C 180,E1 -12124.021,E2 -12124.021} C_VEL
LIN {X 0,Y 383.012,Z 468.774,A -85,B 0,C 180,E1 -12127.336,E2 -12127.336} C_VEL
LIN {X 0,Y 383.064,Z 468.768,A -85,B 0,C 180,E1 -12130.717,E2 -12130.717} C_VEL
LIN {X 0,Y 383.085,Z 468.768,A -85,B 0,C 180,E1 -12134.027,E2 -12134.027} C_VEL
LIN {X 0,Y 383.141,Z 468.757,A -85,B 0,C 180,E1 -12137.284,E2 -12137.284} C_VEL
LIN {X 0,Y 383.155,Z 468.758,A -85,B 0,C 180,E1 -12140.498,E2 -12140.498} C_VEL
LIN {X 0,Y 383.267,Z 468.744,A -85,B 0,C 180,E1 -12143.683,E2 -12143.683} C_VEL
LIN {X 0,Y 383.39,Z 468.73,A -85,B 0,C 180,E1 -12147.899,E2 -12147.899} C_VEL
LIN {X 0,Y 383.522,Z 468.714,A -85,B 0,C 180,E1 -12150,E2 -12150} C_VEL
LIN {X 0,Y 383.251,Z 468.744,A -85,B 0,C 180,E1 -12153.154,E2 -12153.154} C_VEL
LIN {X 0,Y 383.282,Z 468.743,A -85,B 0,C 180,E1 -12156.317,E2 -12156.317} C_VEL
LIN {X 0,Y 383.155,Z 468.757,A -85,B 0,C 180,E1 -12159.502,E2 -12159.502} C_VEL
LIN {X 0,Y 383.13,Z 468.762,A -85,B 0,C 180,E1 -12163.536,E2 -12163.536} C_VEL
LIN {X 0,Y 383.099,Z 468.764,A -85,B 0,C 180,E1 -12167.455,E2 -12167.455} C_VEL
LIN {X 0,Y 383.033,Z 468.771,A -85,B 0,C 180,E1 -12170.647,E2 -12170.647} C_VEL
LIN {X 0,Y 383.038,Z 468.775,A -85,B 0,C 180,E1 -12173.807,E2 -12173.807} C_VEL
LIN {X 0,Y 383.084,Z 468.768,A -85,B 0,C 180,E1 -12176.123,E2 -12176.123} C_VEL
LIN {X 0,Y 382.996,Z 468.779,A -85,B 0,C 180,E1 -12179.7,E2 -12179.7} C_VEL
LIN {X 0,Y 383.016,Z 468.776,A -85,B 0,C 180,E1 -12183.4,E2 -12183.4} C_VEL
LIN {X 0,Y 383.002,Z 468.774,A -85,B 0,C 180,E1 -12185.375,E2 -12185.375} C_VEL
LIN {X 0,Y 382.366,Z 468.859,A -85,B 0,C 180,E1 -12186.253,E2 -12186.253} C_VEL
LIN {X 0,Y 379.57,Z 469.212,A -85,B 0,C 180,E1 -12187.682,E2 -12187.682} C_VEL
LIN {X 0,Y 377.165,Z 469.512,A -85,B 0,C 180,E1 -12188.836,E2 -12188.836} C_VEL
LIN {X 0,Y 376.094,Z 469.641,A -85,B 0,C 180,E1 -12189.728,E2 -12189.728} C_VEL
LIN {X 0,Y 375.987,Z 469.651,A -85,B 0,C 180,E1 -12190.03,E2 -12190.03} C_VEL
LIN {X 0,Y 375.934,Z 469.66,A -85,B 0,C 180,E1 -12193.766,E2 -12193.766} C_VEL
LIN {X 0,Y 375.937,Z 469.655,A -85,B 0,C 180,E1 -12196.811,E2 -12196.811} C_VEL
LIN {X 0,Y 375.965,Z 469.651,A -85,B 0,C 180,E1 -12200.537,E2 -12200.537} C_VEL
LIN {X 0,Y 375.914,Z 469.662,A -85,B 0,C 180,E1 -12203.506,E2 -12203.506} C_VEL
LIN {X 0,Y 375.724,Z 469.686,A -85,B 0,C 180,E1 -12205.864,E2 -12205.864} C_VEL
LIN {X 0,Y 375.363,Z 469.732,A -85,B 0,C 180,E1 -12209.633,E2 -12209.633} C_VEL
LIN {X 0,Y 375.115,Z 469.791,A -85,B 0,C 180,E1 -12212.07,E2 -12212.07} C_VEL
LIN {X 0,Y 374.939,Z 473.233,A -85,B 0,C 180,E1 -12215.645,E2 -12215.645} C_VEL
LIN {X 0,Y 374.878,Z 477.204,A -85,B 0,C 180,E1 -12219.615,E2 -12219.615} C_VEL
LIN {X 0,Y 374.838,Z 479.347,A -85,B 0,C 180,E1 -12221.682,E2 -12221.682} C_VEL
LIN {X 0,Y 377.731,Z 492.929,A -85,B 0,C 180,E1 -12222.373,E2 -12222.373} C_VEL
LIN {X 0,Y 380.032,Z 504.484,A -85,B 0,C 180,E1 -12223.135,E2 -12223.135} C_VEL
LIN {X 0,Y 379.29,Z 516.394,A -85,B 0,C 180,E1 -12224.014,E2 -12224.014} C_VEL
LIN {X 0,Y 378.597,Z 527.21,A -85,B 0,C 180,E1 -12225.027,E2 -12225.027} C_VEL
LIN {X 0,Y 377.764,Z 538.071,A -85,B 0,C 180,E1 -12226.278,E2 -12226.278} C_VEL
LIN {X 0,Y 376.969,Z 547.597,A -85,B 0,C 180,E1 -12227.619,E2 -12227.619} C_VEL
LIN {X 0,Y 376.253,Z 556.838,A -85,B 0,C 180,E1 -12229.234,E2 -12229.234} C_VEL
LIN {X 0,Y 375.692,Z 564.332,A -85,B 0,C 180,E1 -12230.85,E2 -12230.85} C_VEL
LIN {X 0,Y 375.309,Z 570.362,A -85,B 0,C 180,E1 -12232.468,E2 -12232.468} C_VEL
LIN {X 0,Y 375.033,Z 575.121,A -85,B 0,C 180,E1 -12234.084,E2 -12234.084} C_VEL
LIN {X 0,Y 374.808,Z 578.762,A -85,B 0,C 180,E1 -12235.698,E2 -12235.698} C_VEL
LIN {X 0,Y 374.808,Z 580.585,A -85,B 0,C 180,E1 -12236.775,E2 -12236.775} C_VEL
LIN {X 0,Y 374.774,Z 582,A -85,B 0,C 180,E1 -12237.85,E2 -12237.85} C_VEL
LIN {X 0,Y 374.679,Z 583.015,A -85,B 0,C 180,E1 -12238.925,E2 -12238.925} C_VEL
LIN {X 0,Y 374.656,Z 583.579,A -85,B 0,C 180,E1 -12240,E2 -12240} C_VEL
LIN {X 0,Y 374.722,Z 583.727,A -85,B 0,C 180,E1 -12241.074,E2 -12241.074} C_VEL
LIN {X 0,Y 374.82,Z 583.482,A -85,B 0,C 180,E1 -12242.149,E2 -12242.149} C_VEL
LIN {X 0,Y 374.958,Z 582.841,A -85,B 0,C 180,E1 -12243.223,E2 -12243.223} C_VEL
LIN {X 0,Y 375.146,Z 581.747,A -85,B 0,C 180,E1 -12244.297,E2 -12244.297} C_VEL
LIN {X 0,Y 375.18,Z 580.264,A -85,B 0,C 180,E1 -12245.374,E2 -12245.374} C_VEL
LIN {X 0,Y 375.574,Z 577.166,A -85,B 0,C 180,E1 -12247.004,E2 -12247.004} C_VEL
LIN {X 0,Y 376.102,Z 573.088,A -85,B 0,C 180,E1 -12248.597,E2 -12248.597} C_VEL
LIN {X 0,Y 376.74,Z 567.818,A -85,B 0,C 180,E1 -12250.208,E2 -12250.208} C_VEL
LIN {X 0,Y 377.578,Z 561.288,A -85,B 0,C 180,E1 -12251.815,E2 -12251.815} C_VEL
LIN {X 0,Y 378.667,Z 553.155,A -85,B 0,C 180,E1 -12253.415,E2 -12253.415} C_VEL
LIN {X 0,Y 379.507,Z 546.706,A -85,B 0,C 180,E1 -12254.478,E2 -12254.478} C_VEL
LIN {X 0,Y 380.941,Z 535.962,A -85,B 0,C 180,E1 -12255.928,E2 -12255.928} C_VEL
LIN {X 0,Y 382.08,Z 525.326,A -85,B 0,C 180,E1 -12257.116,E2 -12257.116} C_VEL
LIN {X 0,Y 383.308,Z 513.484,A -85,B 0,C 180,E1 -12258.161,E2 -12258.161} C_VEL
LIN {X 0,Y 383.641,Z 508.86,A -85,B 0,C 180,E1 -12258.516,E2 -12258.516} C_VEL
LIN {X 0,Y 380.504,Z 497.072,A -85,B 0,C 180,E1 -12259.612,E2 -12259.612} C_VEL
LIN {X 0,Y 376.398,Z 486.993,A -85,B 0,C 180,E1 -12260.562,E2 -12260.562} C_VEL
LIN {X 0,Y 375.739,Z 484.788,A -85,B 0,C 180,E1 -12260.757,E2 -12260.757} C_VEL
LIN {X 0,Y 375.967,Z 482.661,A -85,B 0,C 180,E1 -12264.283,E2 -12264.283} C_VEL
LIN {X 0,Y 376.312,Z 480.886,A -85,B 0,C 180,E1 -12267.833,E2 -12267.833} C_VEL
LIN {X 0,Y 376.703,Z 479.457,A -85,B 0,C 180,E1 -12271.492,E2 -12271.492} C_VEL
LIN {X 0,Y 377.021,Z 478.801,A -85,B 0,C 180,E1 -12274.002,E2 -12274.002} C_VEL
LIN {X 0,Y 377.307,Z 478.466,A -85,B 0,C 180,E1 -12276.779,E2 -12276.779} C_VEL
LIN {X 0,Y 377.457,Z 478.569,A -85,B 0,C 180,E1 -12279.276,E2 -12279.276} C_VEL
LIN {X 0,Y 377.629,Z 479.16,A -85,B 0,C 180,E1 -12282.066,E2 -12282.066} C_VEL
LIN {X 0,Y 377.871,Z 480.432,A -85,B 0,C 180,E1 -12285.028,E2 -12285.028} C_VEL
LIN {X 0,Y 378.261,Z 482.388,A -85,B 0,C 180,E1 -12288.02,E2 -12288.02} C_VEL
LIN {X 0,Y 378.675,Z 485.323,A -85,B 0,C 180,E1 -12291.215,E2 -12291.215} C_VEL
LIN {X 0,Y 378.714,Z 488.052,A -85,B 0,C 180,E1 -12293.57,E2 -12293.57} C_VEL
LIN {X 0,Y 378.233,Z 491.63,A -85,B 0,C 180,E1 -12296.121,E2 -12296.121} C_VEL
LIN {X 0,Y 377.442,Z 496.108,A -85,B 0,C 180,E1 -12298.929,E2 -12298.929} C_VEL
LIN {X 0,Y 376.663,Z 501.922,A -85,B 0,C 180,E1 -12302.195,E2 -12302.195} C_VEL
LIN {X 0,Y 375.962,Z 508.73,A -85,B 0,C 180,E1 -12305.716,E2 -12305.716} C_VEL
LIN {X 0,Y 375.482,Z 515.972,A -85,B 0,C 180,E1 -12309.188,E2 -12309.188} C_VEL
LIN {X 0,Y 379.069,Z 531.467,A -85,B 0,C 180,E1 -12310.255,E2 -12310.255} C_VEL
LIN {X 0,Y 380.523,Z 541.865,A -85,B 0,C 180,E1 -12311.034,E2 -12311.034} C_VEL
LIN {X 0,Y 381.025,Z 555.328,A -85,B 0,C 180,E1 -12312.142,E2 -12312.142} C_VEL
LIN {X 0,Y 380.153,Z 565.458,A -85,B 0,C 180,E1 -12313.072,E2 -12313.072} C_VEL
LIN {X 0,Y 378.868,Z 576.341,A -85,B 0,C 180,E1 -12314.259,E2 -12314.259} C_VEL
LIN {X 0,Y 377.572,Z 587.294,A -85,B 0,C 180,E1 -12315.738,E2 -12315.738} C_VEL
LIN {X 0,Y 376.601,Z 596.89,A -85,B 0,C 180,E1 -12317.333,E2 -12317.333} C_VEL
LIN {X 0,Y 375.689,Z 604.78,A -85,B 0,C 180,E1 -12318.945,E2 -12318.945} C_VEL
LIN {X 0,Y 375.122,Z 612.165,A -85,B 0,C 180,E1 -12320.837,E2 -12320.837} C_VEL
LIN {X 0,Y 374.77,Z 617.159,A -85,B 0,C 180,E1 -12322.457,E2 -12322.457} C_VEL
LIN {X 0,Y 374.668,Z 620.451,A -85,B 0,C 180,E1 -12323.811,E2 -12323.811} C_VEL
LIN {X 0,Y 374.586,Z 623.853,A -85,B 0,C 180,E1 -12325.696,E2 -12325.696} C_VEL
LIN {X 0,Y 374.553,Z 625.213,A -85,B 0,C 180,E1 -12326.773,E2 -12326.773} C_VEL
LIN {X 0,Y 374.67,Z 626.112,A -85,B 0,C 180,E1 -12327.85,E2 -12327.85} C_VEL
LIN {X 0,Y 374.663,Z 626.588,A -85,B 0,C 180,E1 -12328.925,E2 -12328.925} C_VEL
LIN {X 0,Y 374.665,Z 626.655,A -85,B 0,C 180,E1 -12330,E2 -12330} C_VEL
LIN {X 0,Y 374.671,Z 626.301,A -85,B 0,C 180,E1 -12331.075,E2 -12331.075} C_VEL
LIN {X 0,Y 374.711,Z 625.481,A -85,B 0,C 180,E1 -12332.15,E2 -12332.15} C_VEL
LIN {X 0,Y 374.598,Z 624.229,A -85,B 0,C 180,E1 -12333.226,E2 -12333.226} C_VEL
LIN {X 0,Y 374.679,Z 621.525,A -85,B 0,C 180,E1 -12334.842,E2 -12334.842} C_VEL
LIN {X 0,Y 374.71,Z 617.734,A -85,B 0,C 180,E1 -12336.461,E2 -12336.461} C_VEL
LIN {X 0,Y 374.868,Z 612.775,A -85,B 0,C 180,E1 -12338.083,E2 -12338.083} C_VEL
LIN {X 0,Y 375.181,Z 606.512,A -85,B 0,C 180,E1 -12339.706,E2 -12339.706} C_VEL
LIN {X 0,Y 375.711,Z 598.679,A -85,B 0,C 180,E1 -12341.327,E2 -12341.327} C_VEL
LIN {X 0,Y 376.309,Z 590.707,A -85,B 0,C 180,E1 -12342.676,E2 -12342.676} C_VEL
LIN {X 0,Y 377.109,Z 580.148,A -85,B 0,C 180,E1 -12344.139,E2 -12344.139} C_VEL
LIN {X 0,Y 378.04,Z 569.1,A -85,B 0,C 180,E1 -12345.362,E2 -12345.362} C_VEL
LIN {X 0,Y 378.951,Z 557.007,A -85,B 0,C 180,E1 -12346.429,E2 -12346.429} C_VEL
LIN {X 0,Y 378.785,Z 550.472,A -85,B 0,C 180,E1 -12346.922,E2 -12346.922} C_VEL
LIN {X 0,Y 377.404,Z 538.273,A -85,B 0,C 180,E1 -12347.704,E2 -12347.704} C_VEL
LIN {X 0,Y 375.607,Z 524.363,A -85,B 0,C 180,E1 -12348.381,E2 -12348.381} C_VEL
LIN {X 0,Y 375.181,Z 520.774,A -85,B 0,C 180,E1 -12348.514,E2 -12348.514} C_VEL
LIN {X 0,Y 375.591,Z 513.196,A -85,B 0,C 180,E1 -12351.977,E2 -12351.977} C_VEL
LIN {X 0,Y 376.116,Z 505.688,A -85,B 0,C 180,E1 -12355.453,E2 -12355.453} C_VEL
LIN {X 0,Y 376.818,Z 498.173,A -85,B 0,C 180,E1 -12359.007,E2 -12359.007} C_VEL
LIN {X 0,Y 377.564,Z 490.6,A -85,B 0,C 180,E1 -12362.671,E2 -12362.671} C_VEL
LIN {X 0,Y 378.093,Z 485.519,A -85,B 0,C 180,E1 -12365.186,E2 -12365.186} C_VEL
LIN {X 0,Y 378.121,Z 482.109,A -85,B 0,C 180,E1 -12366.944,E2 -12366.944} C_VEL
LIN {X 0,Y 377.169,Z 476.157,A -85,B 0,C 180,E1 -12370.184,E2 -12370.184} C_VEL
LIN {X 0,Y 376.012,Z 469.756,A -85,B 0,C 180,E1 -12373.847,E2 -12373.847} C_VEL
LIN {X 0,Y 375.995,Z 469.648,A -85,B 0,C 180,E1 -12377.709,E2 -12377.709} C_VEL
LIN {X 0,Y 375.965,Z 469.655,A -85,B 0,C 180,E1 -12380.538,E2 -12380.538} C_VEL
LIN {X 0,Y 375.964,Z 469.652,A -85,B 0,C 180,E1 -12383.496,E2 -12383.496} C_VEL
LIN {X 0,Y 375.961,Z 469.652,A -85,B 0,C 180,E1 -12385.889,E2 -12385.889} C_VEL
LIN {X 0,Y 375.966,Z 469.651,A -85,B 0,C 180,E1 -12389.688,E2 -12389.688} C_VEL
LIN {X 0,Y 376.021,Z 469.645,A -85,B 0,C 180,E1 -12393.348,E2 -12393.348} C_VEL
LIN {X 0,Y 375.998,Z 469.65,A -85,B 0,C 180,E1 -12396.888,E2 -12396.888} C_VEL
LIN {X 0,Y 375.999,Z 469.65,A -85,B 0,C 180,E1 -12400.34,E2 -12400.34} C_VEL
LIN {X 0,Y 376.03,Z 469.643,A -85,B 0,C 180,E1 -12403.719,E2 -12403.719} C_VEL
LIN {X 0,Y 376.105,Z 469.636,A -85,B 0,C 180,E1 -12407.042,E2 -12407.042} C_VEL
LIN {X 0,Y 376.121,Z 469.635,A -85,B 0,C 180,E1 -12410.319,E2 -12410.319} C_VEL
LIN {X 0,Y 376.232,Z 469.622,A -85,B 0,C 180,E1 -12412.487,E2 -12412.487} C_VEL
LIN {X 0,Y 376.173,Z 469.63,A -85,B 0,C 180,E1 -12414.64,E2 -12414.64} C_VEL
LIN {X 0,Y 376.353,Z 469.603,A -85,B 0,C 180,E1 -12417.86,E2 -12417.86} C_VEL
LIN {X 0,Y 376.491,Z 469.587,A -85,B 0,C 180,E1 -12420,E2 -12420} C_VEL
LIN {X 0,Y 376.19,Z 469.623,A -85,B 0,C 180,E1 -12423.213,E2 -12423.213} C_VEL
LIN {X 0,Y 376.236,Z 469.62,A -85,B 0,C 180,E1 -12426.628,E2 -12426.628} C_VEL
LIN {X 0,Y 376.207,Z 469.625,A -85,B 0,C 180,E1 -12428.595,E2 -12428.595} C_VEL
LIN {X 0,Y 376.052,Z 469.641,A -85,B 0,C 180,E1 -12431.864,E2 -12431.864} C_VEL
LIN {X 0,Y 376.061,Z 469.64,A -85,B 0,C 180,E1 -12435.168,E2 -12435.168} C_VEL
LIN {X 0,Y 376.026,Z 469.648,A -85,B 0,C 180,E1 -12438.526,E2 -12438.526} C_VEL
LIN {X 0,Y 375.966,Z 469.654,A -85,B 0,C 180,E1 -12441.954,E2 -12441.954} C_VEL
LIN {X 0,Y 376.008,Z 469.645,A -85,B 0,C 180,E1 -12445.461,E2 -12445.461} C_VEL
LIN {X 0,Y 375.972,Z 469.651,A -85,B 0,C 180,E1 -12449.079,E2 -12449.079} C_VEL
LIN {X 0,Y 375.953,Z 469.653,A -85,B 0,C 180,E1 -12452.829,E2 -12452.829} C_VEL
LIN {X 0,Y 375.961,Z 469.652,A -85,B 0,C 180,E1 -12455.416,E2 -12455.416} C_VEL
LIN {X 0,Y 375.977,Z 469.654,A -85,B 0,C 180,E1 -12458.271,E2 -12458.271} C_VEL
LIN {X 0,Y 375.937,Z 469.655,A -85,B 0,C 180,E1 -12461.601,E2 -12461.601} C_VEL
LIN {X 0,Y 375.931,Z 469.655,A -85,B 0,C 180,E1 -12465.269,E2 -12465.269} C_VEL
LIN {X 0,Y 375.937,Z 469.658,A -85,B 0,C 180,E1 -12468.399,E2 -12468.399} C_VEL
LIN {X 0,Y 375.979,Z 469.652,A -85,B 0,C 180,E1 -12471.729,E2 -12471.729} C_VEL
LIN {X 0,Y 375.983,Z 469.648,A -85,B 0,C 180,E1 -12475.333,E2 -12475.333} C_VEL
LIN {X 0,Y 375.961,Z 469.656,A -85,B 0,C 180,E1 -12478.438,E2 -12478.438} C_VEL
LIN {X 0,Y 375.987,Z 469.653,A -85,B 0,C 180,E1 -12482.141,E2 -12482.141} C_VEL
LIN {X 0,Y 376.01,Z 469.648,A -85,B 0,C 180,E1 -12484.539,E2 -12484.539} C_VEL
LIN {X 0,Y 375.967,Z 469.655,A -85,B 0,C 180,E1 -12488.046,E2 -12488.046} C_VEL
LIN {X 0,Y 376.027,Z 469.644,A -85,B 0,C 180,E1 -12491.474,E2 -12491.474} C_VEL
LIN {X 0,Y 376.063,Z 469.639,A -85,B 0,C 180,E1 -12494.833,E2 -12494.833} C_VEL
LIN {X 0,Y 376.055,Z 469.644,A -85,B 0,C 180,E1 -12498.137,E2 -12498.137} C_VEL
LIN {X 0,Y 376.197,Z 469.626,A -85,B 0,C 180,E1 -12501.947,E2 -12501.947} C_VEL
LIN {X 0,Y 376.167,Z 469.627,A -85,B 0,C 180,E1 -12504.64,E2 -12504.64} C_VEL
LIN {X 0,Y 376.356,Z 469.606,A -85,B 0,C 180,E1 -12507.86,E2 -12507.86} C_VEL
LIN {X 0,Y 376.492,Z 469.59,A -85,B 0,C 180,E1 -12510,E2 -12510} C_VEL
LIN {X 0,Y 376.189,Z 469.624,A -85,B 0,C 180,E1 -12513.213,E2 -12513.213} C_VEL
LIN {X 0,Y 376.24,Z 469.619,A -85,B 0,C 180,E1 -12516.435,E2 -12516.435} C_VEL
LIN {X 0,Y 376.123,Z 469.635,A -85,B 0,C 180,E1 -12519.681,E2 -12519.681} C_VEL
LIN {X 0,Y 376.094,Z 469.638,A -85,B 0,C 180,E1 -12523.658,E2 -12523.658} C_VEL
LIN {X 0,Y 376.049,Z 469.644,A -85,B 0,C 180,E1 -12527.607,E2 -12527.607} C_VEL
LIN {X 0,Y 375.982,Z 469.649,A -85,B 0,C 180,E1 -12530.832,E2 -12530.832} C_VEL
LIN {X 0,Y 375.998,Z 469.649,A -85,B 0,C 180,E1 -12534.281,E2 -12534.281} C_VEL
LIN {X 0,Y 376.024,Z 469.644,A -85,B 0,C 180,E1 -12536.652,E2 -12536.652} C_VEL
LIN {X 0,Y 375.969,Z 469.652,A -85,B 0,C 180,E1 -12540.312,E2 -12540.312} C_VEL
LIN {X 0,Y 375.966,Z 469.655,A -85,B 0,C 180,E1 -12544.111,E2 -12544.111} C_VEL
LIN {X 0,Y 375.958,Z 469.651,A -85,B 0,C 180,E1 -12546.741,E2 -12546.741} C_VEL
LIN {X 0,Y 375.987,Z 469.651,A -85,B 0,C 180,E1 -12550.03,E2 -12550.03} C_VEL
LIN {X 0,Y 375.254,Z 469.741,A -85,B 0,C 180,E1 -12550.923,E2 -12550.923} C_VEL
LIN {X 0,Y 372.346,Z 470.103,A -85,B 0,C 180,E1 -12552.375,E2 -12552.375} C_VEL
LIN {X 0,Y 369.941,Z 470.405,A -85,B 0,C 180,E1 -12553.55,E2 -12553.55} C_VEL
LIN {X 0,Y 368.944,Z 470.525,A -85,B 0,C 180,E1 -12554.458,E2 -12554.458} C_VEL
LIN {X 0,Y 368.88,Z 470.533,A -85,B 0,C 180,E1 -12554.766,E2 -12554.766} C_VEL
LIN {X 0,Y 368.886,Z 470.535,A -85,B 0,C 180,E1 -12558.178,E2 -12558.178} C_VEL
LIN {X 0,Y 368.909,Z 470.532,A -85,B 0,C 180,E1 -12561.36,E2 -12561.36} C_VEL
LIN {X 0,Y 368.859,Z 470.54,A -85,B 0,C 180,E1 -12563.796,E2 -12563.796} C_VEL
LIN {X 0,Y 368.546,Z 470.576,A -85,B 0,C 180,E1 -12567.041,E2 -12567.041} C_VEL
LIN {X 0,Y 368.213,Z 470.621,A -85,B 0,C 180,E1 -12570.247,E2 -12570.247} C_VEL
LIN {X 0,Y 368.106,Z 470.637,A -85,B 0,C 180,E1 -12571.49,E2 -12571.49} C_VEL
LIN {X 0,Y 367.977,Z 471.104,A -85,B 0,C 180,E1 -12572.717,E2 -12572.717} C_VEL
LIN {X 0,Y 367.908,Z 473.428,A -85,B 0,C 180,E1 -12575.149,E2 -12575.149} C_VEL
LIN {X 0,Y 367.796,Z 476.929,A -85,B 0,C 180,E1 -12578.711,E2 -12578.711} C_VEL
LIN {X 0,Y 367.76,Z 479.667,A -85,B 0,C 180,E1 -12581.428,E2 -12581.428} C_VEL
LIN {X 0,Y 370.614,Z 493.029,A -85,B 0,C 180,E1 -12582.123,E2 -12582.123} C_VEL
LIN {X 0,Y 373.086,Z 505.265,A -85,B 0,C 180,E1 -12582.953,E2 -12582.953} C_VEL
LIN {X 0,Y 372.32,Z 516.905,A -85,B 0,C 180,E1 -12583.834,E2 -12583.834} C_VEL
LIN {X 0,Y 371.474,Z 529.408,A -85,B 0,C 180,E1 -12585.05,E2 -12585.05} C_VEL
LIN {X 0,Y 370.679,Z 539.7,A -85,B 0,C 180,E1 -12586.29,E2 -12586.29} C_VEL
LIN {X 0,Y 369.887,Z 548.964,A -85,B 0,C 180,E1 -12587.657,E2 -12587.657} C_VEL
LIN {X 0,Y 369.165,Z 558.052,A -85,B 0,C 180,E1 -12589.303,E2 -12589.303} C_VEL
LIN {X 0,Y 368.585,Z 565.411,A -85,B 0,C 180,E1 -12590.949,E2 -12590.949} C_VEL
LIN {X 0,Y 368.198,Z 571.582,A -85,B 0,C 180,E1 -12592.693,E2 -12592.693} C_VEL
LIN {X 0,Y 367.895,Z 576.598,A -85,B 0,C 180,E1 -12594.519,E2 -12594.519} C_VEL
LIN {X 0,Y 367.737,Z 578.977,A -85,B 0,C 180,E1 -12595.615,E2 -12595.615} C_VEL
LIN {X 0,Y 367.715,Z 580.86,A -85,B 0,C 180,E1 -12596.713,E2 -12596.713} C_VEL
LIN {X 0,Y 367.693,Z 582.309,A -85,B 0,C 180,E1 -12597.809,E2 -12597.809} C_VEL
LIN {X 0,Y 367.613,Z 583.361,A -85,B 0,C 180,E1 -12598.904,E2 -12598.904} C_VEL
LIN {X 0,Y 367.588,Z 584.001,A -85,B 0,C 180,E1 -12600,E2 -12600} C_VEL
LIN {X 0,Y 367.654,Z 584.191,A -85,B 0,C 180,E1 -12601.095,E2 -12601.095} C_VEL
LIN {X 0,Y 367.759,Z 583.986,A -85,B 0,C 180,E1 -12602.19,E2 -12602.19} C_VEL
LIN {X 0,Y 367.91,Z 583.39,A -85,B 0,C 180,E1 -12603.285,E2 -12603.285} C_VEL
LIN {X 0,Y 368.104,Z 582.362,A -85,B 0,C 180,E1 -12604.38,E2 -12604.38} C_VEL
LIN {X 0,Y 368.134,Z 580.917,A -85,B 0,C 180,E1 -12605.477,E2 -12605.477} C_VEL
LIN {X 0,Y 368.543,Z 578.045,A -85,B 0,C 180,E1 -12607.068,E2 -12607.068} C_VEL
LIN {X 0,Y 369.145,Z 573.928,A -85,B 0,C 180,E1 -12608.761,E2 -12608.761} C_VEL
LIN {X 0,Y 369.821,Z 568.788,A -85,B 0,C 180,E1 -12610.401,E2 -12610.401} C_VEL
LIN {X 0,Y 370.723,Z 562.353,A -85,B 0,C 180,E1 -12612.036,E2 -12612.036} C_VEL
LIN {X 0,Y 371.869,Z 554.386,A -85,B 0,C 180,E1 -12613.665,E2 -12613.665} C_VEL
LIN {X 0,Y 372.772,Z 548.065,A -85,B 0,C 180,E1 -12614.745,E2 -12614.745} C_VEL
LIN {X 0,Y 374.131,Z 538.756,A -85,B 0,C 180,E1 -12616.086,E2 -12616.086} C_VEL
LIN {X 0,Y 375.356,Z 528.321,A -85,B 0,C 180,E1 -12617.319,E2 -12617.319} C_VEL
LIN {X 0,Y 376.77,Z 515.938,A -85,B 0,C 180,E1 -12618.488,E2 -12618.488} C_VEL
LIN {X 0,Y 377.222,Z 510.541,A -85,B 0,C 180,E1 -12618.922,E2 -12618.922} C_VEL
LIN {X 0,Y 374.746,Z 500.787,A -85,B 0,C 180,E1 -12619.9,E2 -12619.9} C_VEL
LIN {X 0,Y 370.032,Z 488.825,A -85,B 0,C 180,E1 -12621.1,E2 -12621.1} C_VEL
LIN {X 0,Y 368.785,Z 485.811,A -85,B 0,C 180,E1 -12621.393,E2 -12621.393} C_VEL
LIN {X 0,Y 368.732,Z 485.47,A -85,B 0,C 180,E1 -12621.495,E2 -12621.495} C_VEL
LIN {X 0,Y 369.006,Z 483.614,A -85,B 0,C 180,E1 -12624.772,E2 -12624.772} C_VEL
LIN {X 0,Y 369.384,Z 481.919,A -85,B 0,C 180,E1 -12628.402,E2 -12628.402} C_VEL
LIN {X 0,Y 369.831,Z 480.642,A -85,B 0,C 180,E1 -12632.147,E2 -12632.147} C_VEL
LIN {X 0,Y 370.226,Z 480.04,A -85,B 0,C 180,E1 -12635.287,E2 -12635.287} C_VEL
LIN {X 0,Y 370.512,Z 480.037,A -85,B 0,C 180,E1 -12638.752,E2 -12638.752} C_VEL
LIN {X 0,Y 370.719,Z 480.816,A -85,B 0,C 180,E1 -12642.323,E2 -12642.323} C_VEL
LIN {X 0,Y 370.987,Z 482.264,A -85,B 0,C 180,E1 -12645.498,E2 -12645.498} C_VEL
LIN {X 0,Y 371.389,Z 484.338,A -85,B 0,C 180,E1 -12648.522,E2 -12648.522} C_VEL
LIN {X 0,Y 371.742,Z 487.015,A -85,B 0,C 180,E1 -12651.399,E2 -12651.399} C_VEL
LIN {X 0,Y 371.832,Z 488.546,A -85,B 0,C 180,E1 -12652.783,E2 -12652.783} C_VEL
LIN {X 0,Y 371.404,Z 491.96,A -85,B 0,C 180,E1 -12655.411,E2 -12655.411} C_VEL
LIN {X 0,Y 370.549,Z 496.81,A -85,B 0,C 180,E1 -12658.594,E2 -12658.594} C_VEL
LIN {X 0,Y 369.622,Z 503.094,A -85,B 0,C 180,E1 -12662.235,E2 -12662.235} C_VEL
LIN {X 0,Y 369.02,Z 508.727,A -85,B 0,C 180,E1 -12665.229,E2 -12665.229} C_VEL
LIN {X 0,Y 368.496,Z 515.271,A -85,B 0,C 180,E1 -12668.49,E2 -12668.49} C_VEL
LIN {X 0,Y 372.145,Z 530.339,A -85,B 0,C 180,E1 -12669.622,E2 -12669.622} C_VEL
LIN {X 0,Y 373.939,Z 542.33,A -85,B 0,C 180,E1 -12670.579,E2 -12670.579} C_VEL
LIN {X 0,Y 374.383,Z 555.056,A -85,B 0,C 180,E1 -12671.673,E2 -12671.673} C_VEL
LIN {X 0,Y 374.09,Z 560.948,A -85,B 0,C 180,E1 -12672.224,E2 -12672.224} C_VEL
LIN {X 0,Y 372.702,Z 572.451,A -85,B 0,C 180,E1 -12673.428,E2 -12673.428} C_VEL
LIN {X 0,Y 371.256,Z 583.791,A -85,B 0,C 180,E1 -12674.895,E2 -12674.895} C_VEL
LIN {X 0,Y 370.123,Z 592.54,A -85,B 0,C 180,E1 -12676.269,E2 -12676.269} C_VEL
LIN {X 0,Y 369.162,Z 601.1,A -85,B 0,C 180,E1 -12677.912,E2 -12677.912} C_VEL
LIN {X 0,Y 368.404,Z 608.117,A -85,B 0,C 180,E1 -12679.558,E2 -12679.558} C_VEL
LIN {X 0,Y 367.956,Z 613.82,A -85,B 0,C 180,E1 -12681.211,E2 -12681.211} C_VEL
LIN {X 0,Y 367.66,Z 618.345,A -85,B 0,C 180,E1 -12682.862,E2 -12682.862} C_VEL
LIN {X 0,Y 367.501,Z 621.792,A -85,B 0,C 180,E1 -12684.513,E2 -12684.513} C_VEL
LIN {X 0,Y 367.511,Z 623.548,A -85,B 0,C 180,E1 -12685.613,E2 -12685.613} C_VEL
LIN {X 0,Y 367.465,Z 624.852,A -85,B 0,C 180,E1 -12686.711,E2 -12686.711} C_VEL
LIN {X 0,Y 367.57,Z 625.714,A -85,B 0,C 180,E1 -12687.808,E2 -12687.808} C_VEL
LIN {X 0,Y 367.596,Z 626.165,A -85,B 0,C 180,E1 -12688.904,E2 -12688.904} C_VEL
LIN {X 0,Y 367.595,Z 626.204,A -85,B 0,C 180,E1 -12690,E2 -12690} C_VEL
LIN {X 0,Y 367.604,Z 625.789,A -85,B 0,C 180,E1 -12691.095,E2 -12691.095} C_VEL
LIN {X 0,Y 367.644,Z 624.937,A -85,B 0,C 180,E1 -12692.191,E2 -12692.191} C_VEL
LIN {X 0,Y 367.511,Z 623.653,A -85,B 0,C 180,E1 -12693.289,E2 -12693.289} C_VEL
LIN {X 0,Y 367.612,Z 620.886,A -85,B 0,C 180,E1 -12694.935,E2 -12694.935} C_VEL
LIN {X 0,Y 367.636,Z 617.024,A -85,B 0,C 180,E1 -12696.586,E2 -12696.586} C_VEL
LIN {X 0,Y 367.822,Z 611.992,A -85,B 0,C 180,E1 -12698.239,E2 -12698.239} C_VEL
LIN {X 0,Y 368.144,Z 605.636,A -85,B 0,C 180,E1 -12699.893,E2 -12699.893} C_VEL
LIN {X 0,Y 368.715,Z 597.673,A -85,B 0,C 180,E1 -12701.545,E2 -12701.545} C_VEL
LIN {X 0,Y 369.316,Z 589.584,A -85,B 0,C 180,E1 -12702.92,E2 -12702.92} C_VEL
LIN {X 0,Y 370.085,Z 579.8,A -85,B 0,C 180,E1 -12704.292,E2 -12704.292} C_VEL
LIN {X 0,Y 371.033,Z 568.973,A -85,B 0,C 180,E1 -12705.519,E2 -12705.519} C_VEL
LIN {X 0,Y 371.971,Z 556.966,A -85,B 0,C 180,E1 -12706.605,E2 -12706.605} C_VEL
LIN {X 0,Y 371.5,Z 548.347,A -85,B 0,C 180,E1 -12707.264,E2 -12707.264} C_VEL
LIN {X 0,Y 370.041,Z 535.904,A -85,B 0,C 180,E1 -12708.057,E2 -12708.057} C_VEL
LIN {X 0,Y 368.339,Z 522.631,A -85,B 0,C 180,E1 -12708.69,E2 -12708.69} C_VEL
LIN {X 0,Y 368.101,Z 520.367,A -85,B 0,C 180,E1 -12708.809,E2 -12708.809} C_VEL
LIN {X 0,Y 368.54,Z 512.655,A -85,B 0,C 180,E1 -12712.42,E2 -12712.42} C_VEL
LIN {X 0,Y 369.13,Z 505.195,A -85,B 0,C 180,E1 -12715.97,E2 -12715.97} C_VEL
LIN {X 0,Y 369.889,Z 497.676,A -85,B 0,C 180,E1 -12719.604,E2 -12719.604} C_VEL
LIN {X 0,Y 370.693,Z 489.898,A -85,B 0,C 180,E1 -12723.467,E2 -12723.467} C_VEL
LIN {X 0,Y 371.157,Z 485.059,A -85,B 0,C 180,E1 -12725.944,E2 -12725.944} C_VEL
LIN {X 0,Y 370.817,Z 481.184,A -85,B 0,C 180,E1 -12728.022,E2 -12728.022} C_VEL
LIN {X 0,Y 370.04,Z 476.651,A -85,B 0,C 180,E1 -12730.562,E2 -12730.562} C_VEL
LIN {X 0,Y 368.946,Z 470.53,A -85,B 0,C 180,E1 -12734.15,E2 -12734.15} C_VEL
LIN {X 0,Y 368.941,Z 470.53,A -85,B 0,C 180,E1 -12736.704,E2 -12736.704} C_VEL
LIN {X 0,Y 368.953,Z 470.524,A -85,B 0,C 180,E1 -12739.635,E2 -12739.635} C_VEL
LIN {X 0,Y 368.902,Z 470.533,A -85,B 0,C 180,E1 -12743.144,E2 -12743.144} C_VEL
LIN {X 0,Y 368.897,Z 470.535,A -85,B 0,C 180,E1 -12746.462,E2 -12746.462} C_VEL
LIN {X 0,Y 368.93,Z 470.53,A -85,B 0,C 180,E1 -12749.047,E2 -12749.047} C_VEL
LIN {X 0,Y 368.964,Z 470.528,A -85,B 0,C 180,E1 -12752.797,E2 -12752.797} C_VEL
LIN {X 0,Y 368.946,Z 470.526,A -85,B 0,C 180,E1 -12756.113,E2 -12756.113} C_VEL
LIN {X 0,Y 368.938,Z 470.527,A -85,B 0,C 180,E1 -12759.947,E2 -12759.947} C_VEL
LIN {X 0,Y 368.977,Z 470.521,A -85,B 0,C 180,E1 -12763.399,E2 -12763.399} C_VEL
LIN {X 0,Y 369.059,Z 470.516,A -85,B 0,C 180,E1 -12766.79,E2 -12766.79} C_VEL
LIN {X 0,Y 369.069,Z 470.512,A -85,B 0,C 180,E1 -12770.132,E2 -12770.132} C_VEL
LIN {X 0,Y 369.19,Z 470.499,A -85,B 0,C 180,E1 -12772.342,E2 -12772.342} C_VEL
LIN {X 0,Y 369.146,Z 470.505,A -85,B 0,C 180,E1 -12774.538,E2 -12774.538} C_VEL
LIN {X 0,Y 369.318,Z 470.479,A -85,B 0,C 180,E1 -12777.819,E2 -12777.819} C_VEL
LIN {X 0,Y 369.461,Z 470.463,A -85,B 0,C 180,E1 -12780,E2 -12780} C_VEL
LIN {X 0,Y 369.321,Z 470.482,A -85,B 0,C 180,E1 -12782.181,E2 -12782.181} C_VEL
LIN {X 0,Y 369.206,Z 470.496,A -85,B 0,C 180,E1 -12786.615,E2 -12786.615} C_VEL
LIN {X 0,Y 369.139,Z 470.505,A -85,B 0,C 180,E1 -12788.761,E2 -12788.761} C_VEL
LIN {X 0,Y 369.008,Z 470.52,A -85,B 0,C 180,E1 -12792.093,E2 -12792.093} C_VEL
LIN {X 0,Y 369,Z 470.519,A -85,B 0,C 180,E1 -12795.465,E2 -12795.465} C_VEL
LIN {X 0,Y 368.985,Z 470.522,A -85,B 0,C 180,E1 -12798.893,E2 -12798.893} C_VEL
LIN {X 0,Y 368.935,Z 470.531,A -85,B 0,C 180,E1 -12802.395,E2 -12802.395} C_VEL
LIN {X 0,Y 369.002,Z 470.52,A -85,B 0,C 180,E1 -12805.98,E2 -12805.98} C_VEL
LIN {X 0,Y 368.963,Z 470.525,A -85,B 0,C 180,E1 -12808.812,E2 -12808.812} C_VEL
LIN {X 0,Y 368.901,Z 470.535,A -85,B 0,C 180,E1 -12812.238,E2 -12812.238} C_VEL
LIN {X 0,Y 368.932,Z 470.528,A -85,B 0,C 180,E1 -12815.002,E2 -12815.002} C_VEL
LIN {X 0,Y 368.911,Z 470.532,A -85,B 0,C 180,E1 -12818.641,E2 -12818.641} C_VEL
LIN {X 0,Y 368.884,Z 470.536,A -85,B 0,C 180,E1 -12822.01,E2 -12822.01} C_VEL
LIN {X 0,Y 368.884,Z 470.533,A -85,B 0,C 180,E1 -12825.176,E2 -12825.176} C_VEL
LIN {X 0,Y 368.886,Z 470.538,A -85,B 0,C 180,E1 -12828.178,E2 -12828.178} C_VEL
LIN {X 0,Y 368.913,Z 470.53,A -85,B 0,C 180,E1 -12831.36,E2 -12831.36} C_VEL
LIN {X 0,Y 368.94,Z 470.525,A -85,B 0,C 180,E1 -12835.147,E2 -12835.147} C_VEL
LIN {X 0,Y 368.932,Z 470.527,A -85,B 0,C 180,E1 -12839.047,E2 -12839.047} C_VEL
LIN {X 0,Y 368.967,Z 470.523,A -85,B 0,C 180,E1 -12842.797,E2 -12842.797} C_VEL
LIN {X 0,Y 368.949,Z 470.529,A -85,B 0,C 180,E1 -12846.113,E2 -12846.113} C_VEL
LIN {X 0,Y 368.941,Z 470.53,A -85,B 0,C 180,E1 -12849.947,E2 -12849.947} C_VEL
LIN {X 0,Y 368.98,Z 470.522,A -85,B 0,C 180,E1 -12853.399,E2 -12853.399} C_VEL
LIN {X 0,Y 369.062,Z 470.511,A -85,B 0,C 180,E1 -12856.79,E2 -12856.79} C_VEL
LIN {X 0,Y 369.071,Z 470.514,A -85,B 0,C 180,E1 -12860.132,E2 -12860.132} C_VEL
LIN {X 0,Y 369.183,Z 470.496,A -85,B 0,C 180,E1 -12863.441,E2 -12863.441} C_VEL
LIN {X 0,Y 369.321,Z 470.483,A -85,B 0,C 180,E1 -12867.819,E2 -12867.819} C_VEL
LIN {X 0,Y 369.461,Z 470.466,A -85,B 0,C 180,E1 -12870,E2 -12870} C_VEL
LIN {X 0,Y 369.321,Z 470.482,A -85,B 0,C 180,E1 -12872.181,E2 -12872.181} C_VEL
LIN {X 0,Y 369.2,Z 470.495,A -85,B 0,C 180,E1 -12876.558,E2 -12876.558} C_VEL
LIN {X 0,Y 369.072,Z 470.515,A -85,B 0,C 180,E1 -12879.868,E2 -12879.868} C_VEL
LIN {X 0,Y 369.041,Z 470.517,A -85,B 0,C 180,E1 -12883.772,E2 -12883.772} C_VEL
LIN {X 0,Y 369.005,Z 470.523,A -85,B 0,C 180,E1 -12887.768,E2 -12887.768} C_VEL
LIN {X 0,Y 368.933,Z 470.528,A -85,B 0,C 180,E1 -12891.22,E2 -12891.22} C_VEL
LIN {X 0,Y 368.962,Z 470.523,A -85,B 0,C 180,E1 -12894.775,E2 -12894.775} C_VEL
LIN {X 0,Y 368.967,Z 470.524,A -85,B 0,C 180,E1 -12897.203,E2 -12897.203} C_VEL
LIN {X 0,Y 368.933,Z 470.527,A -85,B 0,C 180,E1 -12900.953,E2 -12900.953} C_VEL
LIN {X 0,Y 368.933,Z 470.527,A -85,B 0,C 180,E1 -12905.001,E2 -12905.001} C_VEL
LIN {X 0,Y 368.913,Z 470.529,A -85,B 0,C 180,E1 -12908.64,E2 -12908.64} C_VEL
LIN {X 0,Y 368.885,Z 470.537,A -85,B 0,C 180,E1 -12912.009,E2 -12912.009} C_VEL
LIN {X 0,Y 368.88,Z 470.533,A -85,B 0,C 180,E1 -12914.766,E2 -12914.766} C_VEL
LIN {X 0,Y 368.252,Z 470.617,A -85,B 0,C 180,E1 -12915.677,E2 -12915.677} C_VEL
LIN {X 0,Y 365.395,Z 470.972,A -85,B 0,C 180,E1 -12917.158,E2 -12917.158} C_VEL
LIN {X 0,Y 362.956,Z 471.274,A -85,B 0,C 180,E1 -12918.356,E2 -12918.356} C_VEL
LIN {X 0,Y 361.915,Z 471.403,A -85,B 0,C 180,E1 -12919.284,E2 -12919.284} C_VEL
LIN {X 0,Y 361.836,Z 471.411,A -85,B 0,C 180,E1 -12919.598,E2 -12919.598} C_VEL
LIN {X 0,Y 361.841,Z 471.41,A -85,B 0,C 180,E1 -12922.978,E2 -12922.978} C_VEL
LIN {X 0,Y 361.634,Z 471.441,A -85,B 0,C 180,E1 -12925.695,E2 -12925.695} C_VEL
LIN {X 0,Y 361.305,Z 471.478,A -85,B 0,C 180,E1 -12928.857,E2 -12928.857} C_VEL
LIN {X 0,Y 360.945,Z 471.529,A -85,B 0,C 180,E1 -12932.14,E2 -12932.14} C_VEL
LIN {X 0,Y 360.85,Z 473.6,A -85,B 0,C 180,E1 -12934.629,E2 -12934.629} C_VEL
LIN {X 0,Y 360.764,Z 475.958,A -85,B 0,C 180,E1 -12937.069,E2 -12937.069} C_VEL
LIN {X 0,Y 360.692,Z 479.504,A -85,B 0,C 180,E1 -12940.656,E2 -12940.656} C_VEL
LIN {X 0,Y 360.719,Z 480.201,A -85,B 0,C 180,E1 -12941.181,E2 -12941.181} C_VEL
LIN {X 0,Y 363.359,Z 492.682,A -85,B 0,C 180,E1 -12941.835,E2 -12941.835} C_VEL
LIN {X 0,Y 366.001,Z 505.546,A -85,B 0,C 180,E1 -12942.724,E2 -12942.724} C_VEL
LIN {X 0,Y 365.343,Z 517.563,A -85,B 0,C 180,E1 -12943.66,E2 -12943.66} C_VEL
LIN {X 0,Y 364.502,Z 529.577,A -85,B 0,C 180,E1 -12944.852,E2 -12944.852} C_VEL
LIN {X 0,Y 363.664,Z 540.247,A -85,B 0,C 180,E1 -12946.163,E2 -12946.163} C_VEL
LIN {X 0,Y 362.748,Z 550.286,A -85,B 0,C 180,E1 -12947.695,E2 -12947.695} C_VEL
LIN {X 0,Y 362.051,Z 559.217,A -85,B 0,C 180,E1 -12949.373,E2 -12949.373} C_VEL
LIN {X 0,Y 361.46,Z 566.389,A -85,B 0,C 180,E1 -12951.051,E2 -12951.051} C_VEL
LIN {X 0,Y 361.047,Z 573.255,A -85,B 0,C 180,E1 -12953.097,E2 -12953.097} C_VEL
LIN {X 0,Y 360.76,Z 577.999,A -85,B 0,C 180,E1 -12954.97,E2 -12954.97} C_VEL
LIN {X 0,Y 360.623,Z 581.111,A -85,B 0,C 180,E1 -12956.648,E2 -12956.648} C_VEL
LIN {X 0,Y 360.614,Z 582.605,A -85,B 0,C 180,E1 -12957.766,E2 -12957.766} C_VEL
LIN {X 0,Y 360.549,Z 583.703,A -85,B 0,C 180,E1 -12958.883,E2 -12958.883} C_VEL
LIN {X 0,Y 360.521,Z 584.403,A -85,B 0,C 180,E1 -12960,E2 -12960} C_VEL
LIN {X 0,Y 360.588,Z 584.654,A -85,B 0,C 180,E1 -12961.117,E2 -12961.117} C_VEL
LIN {X 0,Y 360.7,Z 584.49,A -85,B 0,C 180,E1 -12962.233,E2 -12962.233} C_VEL
LIN {X 0,Y 360.864,Z 583.932,A -85,B 0,C 180,E1 -12963.349,E2 -12963.349} C_VEL
LIN {X 0,Y 361.063,Z 582.983,A -85,B 0,C 180,E1 -12964.465,E2 -12964.465} C_VEL
LIN {X 0,Y 361.092,Z 581.601,A -85,B 0,C 180,E1 -12965.584,E2 -12965.584} C_VEL
LIN {X 0,Y 361.725,Z 577.71,A -85,B 0,C 180,E1 -12967.739,E2 -12967.739} C_VEL
LIN {X 0,Y 362.383,Z 573.275,A -85,B 0,C 180,E1 -12969.488,E2 -12969.488} C_VEL
LIN {X 0,Y 363.427,Z 566.757,A -85,B 0,C 180,E1 -12971.433,E2 -12971.433} C_VEL
LIN {X 0,Y 364.461,Z 559.793,A -85,B 0,C 180,E1 -12973.096,E2 -12973.096} C_VEL
LIN {X 0,Y 365.719,Z 551.205,A -85,B 0,C 180,E1 -12974.751,E2 -12974.751} C_VEL
LIN {X 0,Y 367.475,Z 540.415,A -85,B 0,C 180,E1 -12976.385,E2 -12976.385} C_VEL
LIN {X 0,Y 368.921,Z 529.362,A -85,B 0,C 180,E1 -12977.746,E2 -12977.746} C_VEL
LIN {X 0,Y 370.29,Z 518.492,A -85,B 0,C 180,E1 -12978.823,E2 -12978.823} C_VEL
LIN {X 0,Y 370.871,Z 512.398,A -85,B 0,C 180,E1 -12979.347,E2 -12979.347} C_VEL
LIN {X 0,Y 368.496,Z 503.115,A -85,B 0,C 180,E1 -12980.332,E2 -12980.332} C_VEL
LIN {X 0,Y 365.24,Z 494.445,A -85,B 0,C 180,E1 -12981.279,E2 -12981.279} C_VEL
LIN {X 0,Y 361.891,Z 486.799,A -85,B 0,C 180,E1 -12982.102,E2 -12982.102} C_VEL
LIN {X 0,Y 361.78,Z 486.24,A -85,B 0,C 180,E1 -12982.184,E2 -12982.184} C_VEL
LIN {X 0,Y 362.041,Z 484.6,A -85,B 0,C 180,E1 -12985.282,E2 -12985.282} C_VEL
LIN {X 0,Y 362.481,Z 483.027,A -85,B 0,C 180,E1 -12988.994,E2 -12988.994} C_VEL
LIN {X 0,Y 362.963,Z 481.884,A -85,B 0,C 180,E1 -12992.831,E2 -12992.831} C_VEL
LIN {X 0,Y 363.324,Z 481.474,A -85,B 0,C 180,E1 -12995.665,E2 -12995.665} C_VEL
LIN {X 0,Y 363.519,Z 481.498,A -85,B 0,C 180,E1 -12998.219,E2 -12998.219} C_VEL
LIN {X 0,Y 363.713,Z 482.001,A -85,B 0,C 180,E1 -13001.097,E2 -13001.097} C_VEL
LIN {X 0,Y 363.981,Z 483.237,A -85,B 0,C 180,E1 -13004.404,E2 -13004.404} C_VEL
LIN {X 0,Y 364.342,Z 485.141,A -85,B 0,C 180,E1 -13007.535,E2 -13007.535} C_VEL
LIN {X 0,Y 364.678,Z 487.642,A -85,B 0,C 180,E1 -13010.508,E2 -13010.508} C_VEL
LIN {X 0,Y 364.841,Z 489.332,A -85,B 0,C 180,E1 -13012.166,E2 -13012.166} C_VEL
LIN {X 0,Y 364.584,Z 492.357,A -85,B 0,C 180,E1 -13014.668,E2 -13014.668} C_VEL
LIN {X 0,Y 363.892,Z 496.039,A -85,B 0,C 180,E1 -13017.263,E2 -13017.263} C_VEL
LIN {X 0,Y 362.981,Z 501.415,A -85,B 0,C 180,E1 -13020.609,E2 -13020.609} C_VEL
LIN {X 0,Y 362.196,Z 507.613,A -85,B 0,C 180,E1 -13024.113,E2 -13024.113} C_VEL
LIN {X 0,Y 361.548,Z 514.609,A -85,B 0,C 180,E1 -13027.752,E2 -13027.752} C_VEL
LIN {X 0,Y 362.497,Z 518.286,A -85,B 0,C 180,E1 -13028.037,E2 -13028.037} C_VEL
LIN {X 0,Y 365.189,Z 528.768,A -85,B 0,C 180,E1 -13028.901,E2 -13028.901} C_VEL
LIN {X 0,Y 367.116,Z 539.917,A -85,B 0,C 180,E1 -13029.843,E2 -13029.843} C_VEL
LIN {X 0,Y 367.79,Z 550.233,A -85,B 0,C 180,E1 -13030.747,E2 -13030.747} C_VEL
LIN {X 0,Y 367.605,Z 560.721,A -85,B 0,C 180,E1 -13031.756,E2 -13031.756} C_VEL
LIN {X 0,Y 366.12,Z 572.087,A -85,B 0,C 180,E1 -13032.978,E2 -13032.978} C_VEL
LIN {X 0,Y 364.634,Z 582.513,A -85,B 0,C 180,E1 -13034.345,E2 -13034.345} C_VEL
LIN {X 0,Y 363.418,Z 591.24,A -85,B 0,C 180,E1 -13035.725,E2 -13035.725} C_VEL
LIN {X 0,Y 362.407,Z 599.95,A -85,B 0,C 180,E1 -13037.398,E2 -13037.398} C_VEL
LIN {X 0,Y 361.39,Z 608.115,A -85,B 0,C 180,E1 -13039.353,E2 -13039.353} C_VEL
LIN {X 0,Y 360.894,Z 613.723,A -85,B 0,C 180,E1 -13041.037,E2 -13041.037} C_VEL
LIN {X 0,Y 360.588,Z 618.16,A -85,B 0,C 180,E1 -13042.722,E2 -13042.722} C_VEL
LIN {X 0,Y 360.423,Z 621.534,A -85,B 0,C 180,E1 -13044.405,E2 -13044.405} C_VEL
LIN {X 0,Y 360.416,Z 623.248,A -85,B 0,C 180,E1 -13045.526,E2 -13045.526} C_VEL
LIN {X 0,Y 360.38,Z 624.489,A -85,B 0,C 180,E1 -13046.646,E2 -13046.646} C_VEL
LIN {X 0,Y 360.47,Z 625.32,A -85,B 0,C 180,E1 -13047.765,E2 -13047.765} C_VEL
LIN {X 0,Y 360.53,Z 625.742,A -85,B 0,C 180,E1 -13048.883,E2 -13048.883} C_VEL
LIN {X 0,Y 360.528,Z 625.736,A -85,B 0,C 180,E1 -13050,E2 -13050} C_VEL
LIN {X 0,Y 360.539,Z 625.266,A -85,B 0,C 180,E1 -13051.117,E2 -13051.117} C_VEL
LIN {X 0,Y 360.559,Z 624.381,A -85,B 0,C 180,E1 -13052.234,E2 -13052.234} C_VEL
LIN {X 0,Y 360.426,Z 623.065,A -85,B 0,C 180,E1 -13053.353,E2 -13053.353} C_VEL
LIN {X 0,Y 360.543,Z 620.229,A -85,B 0,C 180,E1 -13055.032,E2 -13055.032} C_VEL
LIN {X 0,Y 360.569,Z 616.288,A -85,B 0,C 180,E1 -13056.716,E2 -13056.716} C_VEL
LIN {X 0,Y 360.801,Z 610.16,A -85,B 0,C 180,E1 -13058.683,E2 -13058.683} C_VEL
LIN {X 0,Y 361.187,Z 603.434,A -85,B 0,C 180,E1 -13060.369,E2 -13060.369} C_VEL
LIN {X 0,Y 361.843,Z 595.109,A -85,B 0,C 180,E1 -13062.052,E2 -13062.052} C_VEL
LIN {X 0,Y 362.541,Z 586.572,A -85,B 0,C 180,E1 -13063.452,E2 -13063.452} C_VEL
LIN {X 0,Y 363.35,Z 576.391,A -85,B 0,C 180,E1 -13064.821,E2 -13064.821} C_VEL
LIN {X 0,Y 364.244,Z 566.029,A -85,B 0,C 180,E1 -13065.959,E2 -13065.959} C_VEL
LIN {X 0,Y 365.003,Z 555.132,A -85,B 0,C 180,E1 -13066.931,E2 -13066.931} C_VEL
LIN {X 0,Y 363.778,Z 542.579,A -85,B 0,C 180,E1 -13067.86,E2 -13067.86} C_VEL
LIN {X 0,Y 362.091,Z 528.722,A -85,B 0,C 180,E1 -13068.657,E2 -13068.657} C_VEL
LIN {X 0,Y 361.051,Z 520.117,A -85,B 0,C 180,E1 -13069.029,E2 -13069.029} C_VEL
LIN {X 0,Y 361.506,Z 512.097,A -85,B 0,C 180,E1 -13072.881,E2 -13072.881} C_VEL
LIN {X 0,Y 362.159,Z 504.64,A -85,B 0,C 180,E1 -13076.509,E2 -13076.509} C_VEL
LIN {X 0,Y 362.747,Z 498.961,A -85,B 0,C 180,E1 -13079.326,E2 -13079.326} C_VEL
LIN {X 0,Y 363.594,Z 491.144,A -85,B 0,C 180,E1 -13083.292,E2 -13083.292} C_VEL
LIN {X 0,Y 364.095,Z 486.245,A -85,B 0,C 180,E1 -13085.834,E2 -13085.834} C_VEL
LIN {X 0,Y 363.909,Z 482.92,A -85,B 0,C 180,E1 -13087.645,E2 -13087.645} C_VEL
LIN {X 0,Y 362.911,Z 477.136,A -85,B 0,C 180,E1 -13090.952,E2 -13090.952} C_VEL
LIN {X 0,Y 361.895,Z 471.407,A -85,B 0,C 180,E1 -13094.447,E2 -13094.447} C_VEL
LIN {X 0,Y 361.884,Z 471.405,A -85,B 0,C 180,E1 -13097.56,E2 -13097.56} C_VEL
LIN {X 0,Y 361.871,Z 471.409,A -85,B 0,C 180,E1 -13100.973,E2 -13100.973} C_VEL
LIN {X 0,Y 361.875,Z 471.41,A -85,B 0,C 180,E1 -13104.655,E2 -13104.655} C_VEL
LIN {X 0,Y 361.838,Z 471.413,A -85,B 0,C 180,E1 -13108.371,E2 -13108.371} C_VEL
LIN {X 0,Y 361.909,Z 471.404,A -85,B 0,C 180,E1 -13112.221,E2 -13112.221} C_VEL
LIN {X 0,Y 361.929,Z 471.404,A -85,B 0,C 180,E1 -13114.71,E2 -13114.71} C_VEL
LIN {X 0,Y 361.893,Z 471.407,A -85,B 0,C 180,E1 -13118.347,E2 -13118.347} C_VEL
LIN {X 0,Y 361.968,Z 471.395,A -85,B 0,C 180,E1 -13122.062,E2 -13122.062} C_VEL
LIN {X 0,Y 361.999,Z 471.392,A -85,B 0,C 180,E1 -13126.101,E2 -13126.101} C_VEL
LIN {X 0,Y 362.033,Z 471.387,A -85,B 0,C 180,E1 -13129.938,E2 -13129.938} C_VEL
LIN {X 0,Y 362.153,Z 471.374,A -85,B 0,C 180,E1 -13132.193,E2 -13132.193} C_VEL
LIN {X 0,Y 362.12,Z 471.38,A -85,B 0,C 180,E1 -13134.431,E2 -13134.431} C_VEL
LIN {X 0,Y 362.282,Z 471.355,A -85,B 0,C 180,E1 -13137.777,E2 -13137.777} C_VEL
LIN {X 0,Y 362.43,Z 471.339,A -85,B 0,C 180,E1 -13140,E2 -13140} C_VEL
LIN {X 0,Y 362.284,Z 471.359,A -85,B 0,C 180,E1 -13142.224,E2 -13142.224} C_VEL
LIN {X 0,Y 362.174,Z 471.373,A -85,B 0,C 180,E1 -13146.686,E2 -13146.686} C_VEL
LIN {X 0,Y 362.076,Z 471.383,A -85,B 0,C 180,E1 -13148.933,E2 -13148.933} C_VEL
LIN {X 0,Y 361.963,Z 471.4,A -85,B 0,C 180,E1 -13152.332,E2 -13152.332} C_VEL
LIN {X 0,Y 361.964,Z 471.399,A -85,B 0,C 180,E1 -13154.621,E2 -13154.621} C_VEL
LIN {X 0,Y 361.962,Z 471.398,A -85,B 0,C 180,E1 -13158.099,E2 -13158.099} C_VEL
LIN {X 0,Y 361.894,Z 471.404,A -85,B 0,C 180,E1 -13161.653,E2 -13161.653} C_VEL
LIN {X 0,Y 361.93,Z 471.399,A -85,B 0,C 180,E1 -13165.29,E2 -13165.29} C_VEL
LIN {X 0,Y 361.92,Z 471.401,A -85,B 0,C 180,E1 -13167.778,E2 -13167.778} C_VEL
LIN {X 0,Y 361.849,Z 471.409,A -85,B 0,C 180,E1 -13171.286,E2 -13171.286} C_VEL
LIN {X 0,Y 361.857,Z 471.413,A -85,B 0,C 180,E1 -13174.281,E2 -13174.281} C_VEL
LIN {X 0,Y 361.867,Z 471.407,A -85,B 0,C 180,E1 -13177.223,E2 -13177.223} C_VEL
LIN {X 0,Y 361.838,Z 471.412,A -85,B 0,C 180,E1 -13180.756,E2 -13180.756} C_VEL
LIN {X 0,Y 361.822,Z 471.417,A -85,B 0,C 180,E1 -13184.368,E2 -13184.368} C_VEL
LIN {X 0,Y 361.839,Z 471.411,A -85,B 0,C 180,E1 -13187.568,E2 -13187.568} C_VEL
LIN {X 0,Y 361.873,Z 471.407,A -85,B 0,C 180,E1 -13190.973,E2 -13190.973} C_VEL
LIN {X 0,Y 361.878,Z 471.407,A -85,B 0,C 180,E1 -13194.655,E2 -13194.655} C_VEL
LIN {X 0,Y 361.841,Z 471.415,A -85,B 0,C 180,E1 -13198.371,E2 -13198.371} C_VEL
LIN {X 0,Y 361.912,Z 471.406,A -85,B 0,C 180,E1 -13202.221,E2 -13202.221} C_VEL
LIN {X 0,Y 361.932,Z 471.4,A -85,B 0,C 180,E1 -13204.71,E2 -13204.71} C_VEL
LIN {X 0,Y 361.896,Z 471.407,A -85,B 0,C 180,E1 -13208.347,E2 -13208.347} C_VEL
LIN {X 0,Y 361.971,Z 471.399,A -85,B 0,C 180,E1 -13212.062,E2 -13212.062} C_VEL
LIN {X 0,Y 362.002,Z 471.395,A -85,B 0,C 180,E1 -13216.101,E2 -13216.101} C_VEL
LIN {X 0,Y 362.035,Z 471.391,A -85,B 0,C 180,E1 -13219.938,E2 -13219.938} C_VEL
LIN {X 0,Y 362.144,Z 471.373,A -85,B 0,C 180,E1 -13223.313,E2 -13223.313} C_VEL
LIN {X 0,Y 362.285,Z 471.359,A -85,B 0,C 180,E1 -13227.777,E2 -13227.777} C_VEL
LIN {X 0,Y 362.431,Z 471.342,A -85,B 0,C 180,E1 -13230,E2 -13230} C_VEL
LIN {X 0,Y 362.285,Z 471.358,A -85,B 0,C 180,E1 -13232.224,E2 -13232.224} C_VEL
LIN {X 0,Y 362.162,Z 471.37,A -85,B 0,C 180,E1 -13236.686,E2 -13236.686} C_VEL
LIN {X 0,Y 362.036,Z 471.39,A -85,B 0,C 180,E1 -13240.062,E2 -13240.062} C_VEL
LIN {X 0,Y 362.002,Z 471.395,A -85,B 0,C 180,E1 -13243.899,E2 -13243.899} C_VEL
LIN {X 0,Y 361.972,Z 471.398,A -85,B 0,C 180,E1 -13247.939,E2 -13247.939} C_VEL
LIN {X 0,Y 361.896,Z 471.407,A -85,B 0,C 180,E1 -13251.653,E2 -13251.653} C_VEL
LIN {X 0,Y 361.933,Z 471.4,A -85,B 0,C 180,E1 -13255.29,E2 -13255.29} C_VEL
LIN {X 0,Y 361.912,Z 471.406,A -85,B 0,C 180,E1 -13257.779,E2 -13257.779} C_VEL
LIN {X 0,Y 361.842,Z 471.414,A -85,B 0,C 180,E1 -13261.629,E2 -13261.629} C_VEL
LIN {X 0,Y 361.878,Z 471.408,A -85,B 0,C 180,E1 -13265.345,E2 -13265.345} C_VEL
LIN {X 0,Y 361.874,Z 471.406,A -85,B 0,C 180,E1 -13269.027,E2 -13269.027} C_VEL
LIN {X 0,Y 361.84,Z 471.41,A -85,B 0,C 180,E1 -13272.829,E2 -13272.829} C_VEL
LIN {X 0,Y 361.822,Z 471.416,A -85,B 0,C 180,E1 -13275.946,E2 -13275.946} C_VEL
LIN {X 0,Y 361.836,Z 471.411,A -85,B 0,C 180,E1 -13279.598,E2 -13279.598} C_VEL
LIN {X 0,Y 361.189,Z 471.492,A -85,B 0,C 180,E1 -13280.527,E2 -13280.527} C_VEL
LIN {X 0,Y 358.353,Z 471.847,A -85,B 0,C 180,E1 -13282.037,E2 -13282.037} C_VEL
